(* CODESYS project DCCM_PLC_3_RECOVERED_2023-01-09T10-26-34.project
   Author: jrfsc
   Version: 0.0.0.0
   Title: DCCM_PLC_3

Project tree, tasks and I/O mapping:
  FdtConnections : FDT Connections, Schneider Electric, version 1.0.0.2
  DCCM_PLC_3 : TM251MESC, Schneider Electric, order no. TM251MESC, version 5.1.9.35
      settings: OPCUA enable = False
    application Application
      libraries: SysTimeRtc, * (System); CAA Memory, * (CAA Technical Workgroup); IecRtsServices, 1.0.4.0 (Schneider Electric)
      task MAST (cyclic, interval 20 ms, priority 15, watchdog 100 ms x 1) calls INPUT_MAPPING, AHU_FAN_CONTROL, AHU_DAMPER_CONTROL, AHU_TEMP_CONTROL, RM1_TERMINAL_LOAD, RM2_TERMINAL_LOAD, RM3_TERMINAL_LOAD, RM4_TERMINAL_LOAD, TEST_VAR, SYSTEM_DATE_TIME, OUTPUT_MAPPING, SR_Main
      program AHU_TEMP_CONTROL [FBD]
      program AHU_FAN_CONTROL [FBD]
      program OUTPUT_MAPPING [ST]
      trace Trace (task MAST): GVL.FAN2_SS
      program RM1_TERMINAL_LOAD [FBD]
      global variables PersistentVars
      global variables GVL
      FBs/
        function block DUTY_CHANGE [ST]
        function block LINEAR [ST]
        function block TERMINAL_LOAD [ST]
        function block SB_HEATING_COOLING [ST]
        function block FB_DEPROX_SP [ST]
        function block MAN_AUTO_STS [ST]
        function block FB_HEATING_OR_COOLING [ST]
        function block FB_SETPOINT_MODE [ST]
        function block FB_FLOATING_VALVE [ST]
        function block FB_OMODE [ST]
        function block FB_9StatesMonitoring [ST]
        function block FB_PMODE [ST]
        function block FB_WATCHDOG [ST]
        function block FB_MAX4 [ST]
        function block FB_DUTY_DUTY_STANDBY_PUMP_SPD [ST]
        function block DUTY [ST]
        function block SATSP_CALC [ST]
      program SYSTEM_DATE_TIME [ST]
      program RM3_TERMINAL_LOAD [FBD]
      Library/
        function block FB_SETPOINT_RAMPING [ST]
      program RM2_TERMINAL_LOAD [FBD]
      LIBRARY/
        function block FB_0_10V_TO_2_10V_OUTPUT [ST]
        function block FB_PULSE_GENERATOR [ST]
        function block FB_2_10V_TO_0_10V_INPUT [ST]
      program SR_Main [FBD]
      program AHU_DAMPER_CONTROL [FBD]
      program TEST_VAR [CFC]
      program RM4_TERMINAL_LOAD [FBD]
      program INPUT_MAPPING [ST]
      Enumeration/
        data type ET_9STATE_MONITORING
        data type ET_OMODE
        data type ET_PMODE
    IO_Bus : IO bus - TM3, Schneider Electric, version 5.1.9.35
      Module_3 : TM3AM6/G, Schneider Electric, order no. TM3AM6/G, version 1.0.0.23
          settings: KPI Configuration.KPI Configuration = 32; KPI Configuration.KPI Configuration = 32; KPI Configuration.KPI Configuration = 0; KPI Configuration.KPI Configuration = 0; KPI Configuration.KPI Configuration = 16; KPI Configuration.KPI Configuration = 39; KPI Configuration.KPI Configuration = 16; KPI Configuration.KPI Configuration = 39; KPI Configuration.KPI Configuration = 16; KPI Configuration.KPI Configuration = 16; KPI Configuration.KPI Configuration = 0; KPI Configuration.KPI Configuration = 0; KPI Configuration.KPI Configuration = 16; KPI Configuration.KPI Configuration = 39; KPI Configuration.KPI Configuration = 16; KPI Configuration.KPI Configuration = 39
          input  iOAD1 : INT  // IW0
          input  iOAD2 : INT  // IW1
          output qOAD1 : INT  // QW0
          output qOAD2 : INT  // QW1
          input  ibModule_3_IBStatusIW0 : BYTE  // IBStatusIW0
          input  ibModule_3_IBStatusIW1 : BYTE  // IBStatusIW1
          input  ibModule_3_IBStatusIW2 : BYTE  // IBStatusIW2
          input  ibModule_3_IBStatusIW3 : BYTE  // IBStatusIW3
          input  ibModule_3_IBStatusQW0 : BYTE  // IBStatusQW0
          input  ibModule_3_IBStatusQW1 : BYTE  // IBStatusQW1
          unmapped channels: IW2, IW3
      Module_4 : TM3AM6/G, Schneider Electric, order no. TM3AM6/G, version 1.0.0.23
          settings: KPI Configuration.KPI Configuration = 32; KPI Configuration.KPI Configuration = 32; KPI Configuration.KPI Configuration = 0; KPI Configuration.KPI Configuration = 0; KPI Configuration.KPI Configuration = 16; KPI Configuration.KPI Configuration = 39; KPI Configuration.KPI Configuration = 16; KPI Configuration.KPI Configuration = 39; KPI Configuration.KPI Configuration = 16; KPI Configuration.KPI Configuration = 16; KPI Configuration.KPI Configuration = 0; KPI Configuration.KPI Configuration = 0; KPI Configuration.KPI Configuration = 16; KPI Configuration.KPI Configuration = 39; KPI Configuration.KPI Configuration = 16; KPI Configuration.KPI Configuration = 39
          input  iSAD1_FB : INT  // IW0
          input  iSAD2_FB : INT  // IW1
          output qSAD1 : INT  // QW0
          output qSAD2 : INT  // QW1
          input  ibModule_4_IBStatusIW0 : BYTE  // IBStatusIW0
          input  ibModule_4_IBStatusIW1 : BYTE  // IBStatusIW1
          input  ibModule_4_IBStatusIW2 : BYTE  // IBStatusIW2
          input  ibModule_4_IBStatusIW3 : BYTE  // IBStatusIW3
          input  ibModule_4_IBStatusQW0 : BYTE  // IBStatusQW0
          input  ibModule_4_IBStatusQW1 : BYTE  // IBStatusQW1
          unmapped channels: IW2, IW3
      Module_1 : TM3AM6/G, Schneider Electric, order no. TM3AM6/G, version 1.0.0.23
          settings: KPI Configuration.KPI Configuration = 32; KPI Configuration.KPI Configuration = 32; KPI Configuration.KPI Configuration = 32; KPI Configuration.KPI Configuration = 32; KPI Configuration.KPI Configuration = 0; KPI Configuration.KPI Configuration = 0; KPI Configuration.KPI Configuration = 0; KPI Configuration.KPI Configuration = 0; KPI Configuration.KPI Configuration = 50; KPI Configuration.KPI Configuration = 0; KPI Configuration.KPI Configuration = 244; KPI Configuration.KPI Configuration = 1; KPI Configuration.KPI Configuration = 50; KPI Configuration.KPI Configuration = 0; KPI Configuration.KPI Configuration = 50; KPI Configuration.KPI Configuration = 0; KPI Configuration.KPI Configuration = 200; KPI Configuration.KPI Configuration = 100; KPI Configuration.KPI Configuration = 200; KPI Configuration.KPI Configuration = 200; KPI Configuration.KPI Configuration = 16; KPI Configuration.KPI Configuration = 16; KPI Configuration.KPI Configuration = 0; KPI Configuration.KPI Configuration = 0; KPI Configuration.KPI Configuration = 16; KPI Configuration.KPI Configuration = 39; KPI Configuration.KPI Configuration = 16; KPI Configuration.KPI Configuration = 39
          input  iSA_VELOCITY : INT  // IW0
          input  iFILTER_DP : INT  // IW1
          input  iOA_VELOCITY2 : INT  // IW2
          input  iOA_VELOCITY1 : INT  // IW3
          output qFAN1_SPD : INT  // QW0
          output qFAN2_SPD : INT  // QW1
          input  ibModule_1_IBStatusIW0 : BYTE  // IBStatusIW0
          input  ibModule_1_IBStatusIW1 : BYTE  // IBStatusIW1
          input  ibModule_1_IBStatusIW2 : BYTE  // IBStatusIW2
          input  ibModule_1_IBStatusIW3 : BYTE  // IBStatusIW3
          input  ibModule_1_IBStatusQW0 : BYTE  // IBStatusQW0
          input  ibModule_1_IBStatusQW1 : BYTE  // IBStatusQW1
      Module_6 : TM3TI8T/G, Schneider Electric, order no. TM3TI8T/G, version 1.0.1.21
          settings: KPI Configuration.KPI Configuration = 81; KPI Configuration.KPI Configuration = 81; KPI Configuration.KPI Configuration = 81; KPI Configuration.KPI Configuration = 81; KPI Configuration.KPI Configuration = 81; KPI Configuration.KPI Configuration = 81; KPI Configuration.KPI Configuration = 81; KPI Configuration.KPI Configuration = 81; KPI Configuration.KPI Configuration = 216; KPI Configuration.KPI Configuration = 254; KPI Configuration.KPI Configuration = 216; KPI Configuration.KPI Configuration = 254; KPI Configuration.KPI Configuration = 216; KPI Configuration.KPI Configuration = 254; KPI Configuration.KPI Configuration = 216; KPI Configuration.KPI Configuration = 254; KPI Configuration.KPI Configuration = 216; KPI Configuration.KPI Configuration = 254; KPI Configuration.KPI Configuration = 216; KPI Configuration.KPI Configuration = 254; KPI Configuration.KPI Configuration = 216; KPI Configuration.KPI Configuration = 254; KPI Configuration.KPI Configuration = 216; KPI Configuration.KPI Configuration = 254; KPI Configuration.KPI Configuration = 220; KPI Configuration.KPI Configuration = 5; KPI Configuration.KPI Configuration = 220; KPI Configuration.KPI Configuration = 5; KPI Configuration.KPI Configuration = 220; KPI Configuration.KPI Configuration = 5; KPI Configuration.KPI Configuration = 220; KPI Configuration.KPI Configuration = 5; KPI Configuration.KPI Configuration = 220; KPI Configuration.KPI Configuration = 5; KPI Configuration.KPI Configuration = 220; KPI Configuration.KPI Configuration = 5; KPI Configuration.KPI Configuration = 220; KPI Configuration.KPI Configuration = 5; KPI Configuration.KPI Configuration = 220; KPI Configuration.KPI Configuration = 5;
            KPI Configuration.KPI Configuration = 16; KPI Configuration.KPI Configuration = 39; KPI Configuration.KPI Configuration = 137; KPI Configuration.KPI Configuration = 15; KPI Configuration.KPI Configuration = 16; KPI Configuration.KPI Configuration = 39; KPI Configuration.KPI Configuration = 137; KPI Configuration.KPI Configuration = 15; KPI Configuration.KPI Configuration = 16; KPI Configuration.KPI Configuration = 39; KPI Configuration.KPI Configuration = 137; KPI Configuration.KPI Configuration = 15; KPI Configuration.KPI Configuration = 16; KPI Configuration.KPI Configuration = 39; KPI Configuration.KPI Configuration = 137; KPI Configuration.KPI Configuration = 15; KPI Configuration.KPI Configuration = 16; KPI Configuration.KPI Configuration = 39; KPI Configuration.KPI Configuration = 137; KPI Configuration.KPI Configuration = 15; KPI Configuration.KPI Configuration = 16; KPI Configuration.KPI Configuration = 39; KPI Configuration.KPI Configuration = 137; KPI Configuration.KPI Configuration = 15; KPI Configuration.KPI Configuration = 16; KPI Configuration.KPI Configuration = 39; KPI Configuration.KPI Configuration = 137; KPI Configuration.KPI Configuration = 15; KPI Configuration.KPI Configuration = 16; KPI Configuration.KPI Configuration = 39; KPI Configuration.KPI Configuration = 137; KPI Configuration.KPI Configuration = 15
          input  iSAT : INT  // IW0
          input  iRAT : INT  // IW1
          input  iOCT : INT  // IW2
          input  iOAT : INT  // IW3
          input  iRMT1 : INT  // IW4
          input  iRMT2 : INT  // IW5
          input  iRMT3 : INT  // IW6
          input  iRMT4 : INT  // IW7
          input  ibModule_6_IBStatusIW0 : BYTE  // IBStatusIW0
          input  ibModule_6_IBStatusIW1 : BYTE  // IBStatusIW1
          input  ibModule_6_IBStatusIW2 : BYTE  // IBStatusIW2
          input  ibModule_6_IBStatusIW3 : BYTE  // IBStatusIW3
          input  ibModule_6_IBStatusIW4 : BYTE  // IBStatusIW4
          input  ibModule_6_IBStatusIW5 : BYTE  // IBStatusIW5
          input  ibModule_6_IBStatusIW6 : BYTE  // IBStatusIW6
          input  ibModule_6_IBStatusIW7 : BYTE  // IBStatusIW7
      Module_2 : TM3AM6/G, Schneider Electric, order no. TM3AM6/G, version 1.0.0.23
          settings: KPI Configuration.KPI Configuration = 32; KPI Configuration.KPI Configuration = 32; KPI Configuration.KPI Configuration = 32; KPI Configuration.KPI Configuration = 0; KPI Configuration.KPI Configuration = 0; KPI Configuration.KPI Configuration = 0; KPI Configuration.KPI Configuration = 16; KPI Configuration.KPI Configuration = 39; KPI Configuration.KPI Configuration = 16; KPI Configuration.KPI Configuration = 39; KPI Configuration.KPI Configuration = 244; KPI Configuration.KPI Configuration = 1; KPI Configuration.KPI Configuration = 200; KPI Configuration.KPI Configuration = 16; KPI Configuration.KPI Configuration = 16; KPI Configuration.KPI Configuration = 0; KPI Configuration.KPI Configuration = 0; KPI Configuration.KPI Configuration = 16; KPI Configuration.KPI Configuration = 39; KPI Configuration.KPI Configuration = 16; KPI Configuration.KPI Configuration = 39
          input  iFAN1_SPDFB : INT  // IW0
          input  iFAN2_SPDFB : INT  // IW1
          input  iFILTER2_DP : INT  // IW2
          output qAHU_HV : INT  // QW0
          output qAHU_CV : INT  // QW1
          input  ibModule_2_IBStatusIW0 : BYTE  // IBStatusIW0
          input  ibModule_2_IBStatusIW1 : BYTE  // IBStatusIW1
          input  ibModule_2_IBStatusIW2 : BYTE  // IBStatusIW2
          input  ibModule_2_IBStatusIW3 : BYTE  // IBStatusIW3
          input  ibModule_2_IBStatusQW0 : BYTE  // IBStatusQW0
          input  ibModule_2_IBStatusQW1 : BYTE  // IBStatusQW1
          unmapped channels: IW3
      Module_5 : TM3DM24R/G, Schneider Electric, order no. TM3DM24R/G, version 1.0.2.0
          input  iFAN1_RUN : BOOL  // IW0.I0
          input  iFAN1_FAULT : BOOL  // IW0.I1
          input  iFAN1_READY : BOOL  // IW0.I2
          input  iFAN2_RUN : BOOL  // IW0.I3
          input  iFAN2_FAULT : BOOL  // IW0.I4
          input  iFAN2_READY : BOOL  // IW0.I5
          input  iRAD1_2_STS : BOOL  // IW0.I6
          input  iFIRE_DAMPER_STS : BOOL  // IW0.I7
          input  iDUCT_SMOKE_DETECTOR : BOOL  // IW0.I8
          input  iFAN1_MANUAL_SW : BOOL  // IW0.I12
          input  iFAN1_AUTO_SW : BOOL  // IW0.I13
          input  iFAN2_MANUAL_SW : BOOL  // IW0.I14
          input  iFAN2_AUTO_SW : BOOL  // IW0.I15
          output qFAN1_SS : BOOL  // QB0.Q0
          output qFAN2_SS : BOOL  // QB0.Q1
          output qFAN1_RAD1_2 : BOOL  // QB0.Q2
          output qISO_NORMAL_MODE : BOOL  // QB0.Q3
          unmapped channels: IW0, QB0
    Serial_Line_1 : Serial line, Schneider Electric, version 5.1.9.35
      Machine_Expert_Network_Manager : Machine Expert-Network Manager, Schneider Electric, version 4.0.0.4
    CAN_1 : CANopen bus, Schneider Electric, version 5.1.9.35
    COM_Bus : COM bus, Schneider Electric, version 5.1.9.35
    Ethernet_1 : Ethernet Network, Schneider Electric, version 5.1.9.35
        settings: WebServer = TRUE; FTP Server = FALSE; SoMachine Protocol = TRUE; Modbus Server = TRUE; NetManage Protocol = TRUE; SNMP protocol = FALSE; WebVisu protocol = FALSE; Secured Web Server = TRUE
*)

// DCCM_PLC_3/Application/Enumeration/ET_9STATE_MONITORING
{attribute 'qualified_only' := ''}
{attribute 'strict' := ''}
TYPE ET_9STATE_MONITORING :
(
	STOPPED := 0,
	RUNNING := 1,
	STARTING := 2,
	STOPPING := 3,
	START_FAIL := 4,
	STOP_FAIL := 5,
	UNEXPECTED_START := 6,
	UNEXPECTED_STOP := 7,
	FIRE_STOP := 8,
	UNKNOWN := 9
);
END_TYPE

// DCCM_PLC_3/Application/Enumeration/ET_OMODE
{attribute 'qualified_only' := ''}
{attribute 'strict' := ''}
TYPE ET_OMODE :
(
	UNOCC := 0,
	OPTSTART := 1,
	SCH := 2,
	AHRS := 3,
	MOTDETECT := 4,
	SETBACK := 7
);
END_TYPE

// DCCM_PLC_3/Application/Enumeration/ET_PMODE
{attribute 'qualified_only' := ''}
{attribute 'strict' := ''}
TYPE ET_PMODE :
(
	OFF_NORMAL := 0,
	OFF_PCMS := 1,
	OFF_Fire := 2,
	OFF_DMPRLOCK := 3,
	OFF_RESET := 4,
	Startup := 5,
	Purge := 6,
	RUN_NORMAL := 7
);
END_TYPE

// DCCM_PLC_3/Application/PersistentVars
{attribute 'qualified_only'}
VAR_GLOBAL PERSISTENT RETAIN
	// Generated instance path of persistent variable
	GVL.RM1_RMTSP: REAL := 22.0;
	// Generated instance path of persistent variable
	GVL.RM2_RMTSP: REAL := 22.0;
	// Generated instance path of persistent variable
	GVL.RM3_RMTSP: REAL := 22.0;
	// Generated instance path of persistent variable
	GVL.FAN1_SPD_MAN: REAL;
	// Generated instance path of persistent variable
	GVL.SA_VELOCITY_SP: REAL := 35.0;
	// Generated instance path of persistent variable
	GVL.FILTER_DPSP: REAL := 100.0;
	// Generated instance path of persistent variable
	GVL.SATSP_MAX: REAL := 30.0;
	// Generated instance path of persistent variable
	GVL.SATSP_MIN: REAL := 12.0;
	// Generated instance path of persistent variable
	GVL.SATSP_MID: REAL := 20.0;
	// Generated instance path of persistent variable
	GVL.AHU_POAD_SP: REAL := 0.0;
	// Generated instance path of persistent variable
	GVL.AHU_OAD_SP: REAL := 100.0;
	// Generated instance path of persistent variable
	GVL.FILTER2_DP_ALMSP: REAL := 350.0;
	// Generated instance path of persistent variable
	GVL.FAN_DEPROX1_SP: REAL := 18.0;
	// Generated instance path of persistent variable
	GVL.FAN_DEPROX2_SP: REAL := 1.0;
	// Generated instance path of persistent variable
	GVL.FAN_DEPROX4_SPDSP: REAL := 0.0;
	// Generated instance path of persistent variable
	GVL.FAN_DEPROX4_SP: REAL := 0.0;
END_VAR

// DCCM_PLC_3/Application/GVL
{attribute 'qualified_only'}
VAR_GLOBAL
	AHU_RAD_MAN AT %MD550: REAL;
	AHU_RAD_MD AT %MX5.6: bool;
	FAN1_SPD AT %MD500: REAL;
	FAN2_SPD AT %MD501: REAL;
	SA_VELOCITY AT %MD502: REAL;
	FILTER_DP AT %MD503: REAL;
	OA_VELOCITY1 AT %MD504: REAL;
	OA_VELOCITY2 AT %MD505: REAL;
	AHU_HV AT %MD506: REAL;
	AHU_CV AT %MD507: REAL;
	FAN1_SPDFB AT %MD508: REAL;
	FAN2_SPDFB AT %MD509: REAL;
	OAD AT %MD510: REAL;
	SAD1 AT %MD512: REAL;
	SAD2 AT %MD513: REAL;
	FAN1_RUN AT %MX0.0: BOOL;
	FAN1_FAULT AT %MX0.1: BOOL;
	FAN1_READY AT %MX0.2: BOOL;
	FAN2_RUN AT %MX0.3: BOOL;
	FAN2_FAULT AT %MX0.4: BOOL;
	FAN2_READY AT %MX0.5: BOOL;
	RAD1_2_STS AT %MX0.6: BOOL;
	FIRE_DAMPER_STS AT %MX0.7: BOOL;
	DUCT_SMOKE_DETECTOR AT %MX1.0: BOOL;
	FAN1_MANUAL_SW AT %MX1.1: BOOL;
	FAN1_AUTO_SW AT %MX1.2: BOOL;
	FAN2_MANUAL_SW AT %MX1.3: BOOL;
	FAN2_AUTO_SW AT %MX1.4: BOOL;
	FAN1_SS AT %MX1.5: BOOL;
	FAN2_SS AT %MX1.6: BOOL;
	FAN1_RAD1_2 AT %MX1.7: BOOL;
	// NEED TO FIGURE OUT WHAT THIS DOES
	ISO_NORMAL_MODE AT %MX2.0: BOOL;
	SAT AT %MD514: REAL;
	RAT AT %MD515: REAL;
	OCT AT %MD516: REAL;
	OAT AT %MD517: REAL;
	RMT1 AT %MD518: REAL;
	RMT2 AT %MD519: REAL;
	RMT3 AT %MD520: REAL;
	RMT4 AT %MD521: REAL;
END_VAR
VAR_GLOBAL RETAIN PERSISTENT
	RM1_RMTSP AT %MD522: REAL := 22;
	RM2_RMTSP AT %MD523: REAL := 22;
	RM3_RMTSP AT %MD524: REAL := 22;
END_VAR
VAR_GLOBAL RETAIN
	RM4_RMTSP AT %MD525: REAL := 22;
END_VAR
VAR_GLOBAL PERSISTENT
	FAN1_SPD_MAN AT %MD526: REAL;
END_VAR
VAR_GLOBAL
	FAN1_SPD_MD AT %MX2.1: BOOL := TRUE;
	FAN2_SPD_MAN AT %MD527: REAL;
	FAN2_SPD_MD AT %MX2.2: BOOL := TRUE;
END_VAR
VAR_GLOBAL RETAIN PERSISTENT
	SA_VELOCITY_SP AT %MD528: REAL := 35;
	FILTER_DPSP AT %MD529: REAL := 100;
END_VAR
VAR_GLOBAL
	FILTER_DP_ALM AT %MX2.3: BOOL;
	AHU_HV_MAN AT %MD530: REAL;
	AHU_HV_MD AT %MX2.4: BOOL := TRUE;
	AHU_CV_MAN AT %MD531: REAL;
	AHU_CV_MD AT %MX2.5: BOOL := TRUE;
	OAD_MAN AT %MD532: REAL;
	OAD_MD AT %MX2.6: BOOL := TRUE;
	SAD1_MAN AT %MD534: REAL;
	SAD1_MD AT %MX3.0: BOOL := TRUE;
	SAD2_MAN AT %MD535: REAL;
	SAD2_MD AT %MX3.1: BOOL := TRUE;
	FAN1_SS_MAN AT %MX3.2: BOOL;
	FAN1_SS_MD AT %MX3.3: BOOL := TRUE;
	FAN2_SS_MAN AT %MX3.4: BOOL;
	FAN2_SS_MD AT %MX3.5: BOOL := TRUE;
	RM1_TL AT %MD536: REAL;
	RM2_TL AT %MD537: REAL;
	RM3_TL AT %MD538: REAL;
	RM4_TL AT %MD539: REAL;
	TL AT %MD540: REAL;
	SATSP AT %MD541: REAL;
	SATSP_MAN AT %MD542: REAL;
	SATSP_MD AT %MX3.6: BOOL := TRUE;
END_VAR
VAR_GLOBAL RETAIN PERSISTENT
	SATSP_MAX AT %MD543: REAL := 30;
	SATSP_MIN AT %MD544: REAL := 12;
END_VAR
VAR_GLOBAL
	FAN_DUTY AT %MX3.7: BOOL;
	FAN_DUTY_MAN AT %MX4.0: BOOL;
	FAN_DUTY_MD AT %MX4.1: BOOL := TRUE;
	SYS_DAY: UINT;
	SYS_HOUR: UINT;
	SYS_MINUTE: UINT;
	FAN1_STS AT %MW9000: UINT;
	FAN2_STS AT %MW9001: UINT;
	FAN1_RAD1_2_MAN AT %MX6.4: BOOL;
	FAN1_RAD1_2_MD AT %MX4.2: BOOL := TRUE;
	MAX_TL AT %MD546: REAL;
	FAN2_DISCHARGE_DAMPER AT %MX5.3: BOOL;
END_VAR
VAR_GLOBAL RETAIN PERSISTENT
	SATSP_MID AT %MD547: REAL := 20;
END_VAR
VAR_GLOBAL
	PANDEMIC_MODE AT %MX4.3: BOOL;
	FAN1_DISCHARGE_DAMPER AT %MX5.0: BOOL;
	FAN1_DISCHARGE_DAMPER_MD AT %MX5.1: BOOL := TRUE;
	FAN2_DISCHARGE_DAMPER_MD AT %MX5.4: BOOL := TRUE;
	FAN2_DISCHARGE_DAMPER_MAN AT %MX5.5: BOOL;
	FAN1_DISCHARGE_DAMPER_MAN AT %MX5.2: BOOL;
	EAD AT %MD548: REAL;
	AHU_RAD AT %MD549: REAL;
	FAN1_DISCHARGE_DAMPER_STS AT %MX5.7: BOOL;
	FAN2_DISCHARGE_DAMPER_STS AT %MX6.0: BOOL;
	POAD_MAN AT %MD559: REAL;
END_VAR
VAR_GLOBAL RETAIN PERSISTENT
	AHU_POAD_SP AT %MD554: REAL := 0;
END_VAR
VAR_GLOBAL
	POAD_MD AT %MX6.2: BOOL := TRUE;
	POAD AT %MD555: REAL;
	OAD_VELOCITY AT %MD556: REAL;
	OAP_VELOCITY AT %MD557: REAL;
	OAD_STS AT %MD560: REAL;
	OAP_STS AT %MD561: REAL;
END_VAR
VAR_GLOBAL RETAIN PERSISTENT
	AHU_OAD_SP AT %MD558: REAL := 100;
END_VAR
VAR_GLOBAL
	FAN1_DAMPER_STS AT %MD562: REAL;
	FAN2_DAMPER_STS AT %MD563: REAL;
	OAD1_FB AT %MD550: REAL;
	OAD2_FB AT %MD551: REAL;
	SAD1_FB AT %MD552: REAL;
	SAD2_FB AT %MD553: REAL;
	PAN_MODE_OK AT %MX6.1: BOOL;
	OAD_LS AT %MD564: REAL;
	POAD_LS AT %MD565: REAL;
	SAD_LS AT %MD566: REAL;
	FAN1_SW_STS AT %MW9002: INT;
	FAN2_SW_STS AT %MW9003: INT;
	FILTER2_DP AT %MD567: REAL;
END_VAR
VAR_GLOBAL RETAIN PERSISTENT
	FILTER2_DP_ALMSP AT %MD568: REAL := 350;
END_VAR
VAR_GLOBAL
	FILTER2_DP_ALM AT %MX6.3: BOOL;
END_VAR
VAR_GLOBAL RETAIN PERSISTENT
	FAN_DEPROX1_SP AT %MD569: REAL := 18;
	FAN_DEPROX2_SP AT %MD570: REAL := 1;
	FAN_DEPROX4_SPDSP AT %MD571: REAL := 0;
END_VAR
VAR_GLOBAL
	ROOM1_DEPROX: INT;
	ROOM2_DEPROX: INT;
	ROOM3_DEPROX: INT;
	ROOM4_DEPROX: INT;
END_VAR
VAR_GLOBAL RETAIN PERSISTENT
	FAN_DEPROX4_SP AT %MD571: REAL := 0;
END_VAR
VAR_GLOBAL
	SAD1_ALM AT %MX6.4: BOOL;
	SAD2_ALM AT %MX6.5: BOOL;
	OAD_ALM AT %MX6.6: BOOL;
	POAD_ALM AT %MX6.7: BOOL;
	RAD_ALM AT %MX7.0: BOOL;
	PAND_ALM AT %MX7.1: BOOL;
	SEND_PAND_ALM AT %MW9004: INT;
	OAD_L2_SP AT %MD572: REAL;
	POAD_L2_SP AT %MD573: REAL;
	SA_L2_SP AT %MD574: REAL;
	FAN1_DIG_FLT AT %MX7.2: BOOL;
	FAN2_DIG_FLT AT %MX7.3: BOOL;
	FAN2_FLT_RESET AT %MX7.4: BOOL;
	FAN1_FLT_RESET AT %MX7.5: BOOL;
END_VAR

// DCCM_PLC_3/Application/INPUT_MAPPING
PROGRAM INPUT_MAPPING
VAR
	BELIMO_IP: FB_2_10V_TO_0_10V_INPUT;
END_VAR

//MAPPING HARDWARE INPUTS TO MEMORY WORDS

GVL.SA_VELOCITY := TO_REAL(iSA_VELOCITY);					//MODULE 1 TM3AM6 INPUT 0
GVL.FILTER_DP := TO_REAL(iFILTER_DP);						//MODULE 1 TM3AM6 INPUT 1
//GVL.OA_VELOCITY1 := TO_REAL(iOA_VELOCITY1);	LOOK AT BOTTOM OF MAPPING				//MODULE 1 TM3AM6 INPUT 2
//GVL.OA_VELOCI0TY2 := TO_REAL(iOA_VELOCITY2);					//MODULE 1 TM3AM6 INPUT 3

GVL.FAN1_SPDFB := TO_REAL(iFAN1_SPDFB) / 100;						//MODULE 2 TM3AM6 INPUT 0
GVL.FAN2_SPDFB := TO_REAL(iFAN2_SPDFB) / 100;						//MODULE 2 TM3AM6 INPUT 1

//GVL.OAD1_FB := TO_REAL(iOAD1);		 LOOK AT BOTTOM OF MAPPING		//MODULE 3 TM3AM6 INPUT 0
//GVL.OAD2_FB := TO_REAL(iOAD2);								//MODULE 3 TM3AM6 INPUT 1

GVL.SAD1_FB := TO_REAL(iSAD1_FB);							//MODULE 4 TM3AM6 INPUT 0
GVL.SAD2_FB := TO_REAL(iSAD2_FB);							//MODULE 4 TM3AM6 INPUT 1

GVL.FAN1_RUN := iFAN1_RUN;									//MODULE 5 TM3DM24R INPUT 0
GVL.FAN1_FAULT := iFAN1_FAULT;								//MODULE 5 TM3DM24R INPUT 1
GVL.FAN1_READY := iFAN1_READY;								//MODULE 5 TM3DM24R INPUT 2
GVL.FAN2_RUN := iFAN2_RUN;									//MODULE 5 TM3DM24R INPUT 3
GVL.FAN2_FAULT := iFAN2_FAULT;								//MODULE 5 TM3DM24R INPUT 4
GVL.FAN2_READY := iFAN2_READY;								//MODULE 5 TM3DM24R INPUT 5
GVL.RAD1_2_STS := NOT(iRAD1_2_STS);								//MODULE 5 TM3DM24R INPUT 6
GVL.FIRE_DAMPER_STS := iFIRE_DAMPER_STS;					//MODULE 5 TM3DM24R INPUT 7
GVL.DUCT_SMOKE_DETECTOR := iDUCT_SMOKE_DETECTOR;			//MODULE 5 TM3DM24R INPUT 8

GVL.FAN1_MANUAL_SW := iFAN1_MANUAL_SW;						//MODULE 5 TM3DM24R INPUT 12
GVL.FAN1_AUTO_SW := iFAN1_AUTO_SW;							//MODULE 5 TM3DM24R INPUT 13
GVL.FAN2_MANUAL_SW := iFAN2_MANUAL_SW;						//MODULE 5 TM3DM24R INPUT 14
GVL.FAN2_AUTO_SW := iFAN2_AUTO_SW;							//MODULE 5 TM3DM24R INPUT 15

GVL.SAT := TO_REAL(iSAT) / 10.0;											//MODULE 6 TM3TI8T INPUT 0
GVL.RAT := TO_REAL(iRAT) / 10.0;											//MODULE 6 TM3TI8T INPUT 1
GVL.OCT := TO_REAL(iOCT) / 10.0;											//MODULE 6 TM3TI8T INPUT 2
GVL.OAT := TO_REAL(iOAT) / 10.0;											//MODULE 6 TM3TI8T INPUT 3
GVL.RMT1 := TO_REAL(iRMT1) / 10.0;											//MODULE 6 TM3TI8T INPUT 4
GVL.RMT2 := TO_REAL(iRMT2) / 10.0;											//MODULE 6 TM3TI8T INPUT 5
GVL.RMT3 := TO_REAL(iRMT3) / 10.0;											//MODULE 6 TM3TI8T INPUT 6
GVL.RMT4 := TO_REAL(iRMT4) / 10.0;											//MODULE 6 TM3TI8T INPUT 7

//To be assigned
GVL.OAD_VELOCITY := TO_REAL(iOA_VELOCITY1);	 //Outside Air Velocity from OA Damper
GVL.OAP_VELOCITY := TO_REAL(iOA_VELOCITY2);	 //Outside Air Velocity from OA Pandemic Mode Damper
BELIMO_IP(IN_PRCT := (TO_REAL(iOAD1) / 100));
GVL.OAD_STS := 100 - BELIMO_IP.OUT_PRCT;				 //OA Damper FEEDBACK
BELIMO_IP(IN_PRCT := (TO_REAL(iOAD2) / 100));
GVL.OAP_STS := 100 - BELIMO_IP.OUT_PRCT;			     //OA Pandemic Mode Damper FEEDBACK

BELIMO_IP(IN_PRCT := TO_REAL(iSAD1_FB) / 100);
GVL.FAN1_DAMPER_STS := 100 - BELIMO_IP.OUT_PRCT;	//FAN1 Damper
BELIMO_IP(IN_PRCT := TO_REAL(iSAD2_FB) / 100);
GVL.FAN2_DAMPER_STS := 100 - BELIMO_IP.OUT_PRCT;	//FAN2 Damper

GVL.FILTER2_DP := TO_REAL(iFILTER2_DP);				//SECOND FILTER DP

GVL.OAD_LS := GVL.OAD_VELOCITY * 19.5;					//OAD VP IN L/S
GVL.POAD_LS := GVL.OAP_VELOCITY * 63;				//OAP VP IN L/S
GVL.SAD_LS := GVL.SA_VELOCITY * 25.21;						//SAD VP L/S

GVL.SEND_PAND_ALM := TO_INT(GVL.PANDEMIC_MODE);


GVL.SA_L2_SP := GVL.SA_VELOCITY_SP * 25.21;

END_PROGRAM

// DCCM_PLC_3/Application/LIBRARY/FB_2_10V_TO_0_10V_INPUT
FUNCTION_BLOCK FB_2_10V_TO_0_10V_INPUT
VAR_INPUT
	/// 0-10V = 0-100%
	IN_PRCT: REAL;
END_VAR
VAR_OUTPUT
	/// 2-10V = 0-100%
	OUT_PRCT: REAL;
END_VAR
VAR
	result: REAL;
	LIN: LINEAR;
END_VAR

LIN (X1:=2, Y1:=0, X2:=10, Y2:=10, INPUT:= IN_PRCT/10);
OUT_PRCT := MAX(0, MIN(LIN.OUTPUT * 10, 100));

END_FUNCTION_BLOCK

// DCCM_PLC_3/Application/FBs/LINEAR
FUNCTION_BLOCK LINEAR
VAR_INPUT
	INPUT: REAL;
	X1: REAL;
	Y1: REAL;
	X2: REAL;
	Y2: REAL;
END_VAR
VAR
	M: REAL;
END_VAR
VAR_OUTPUT
	OUTPUT: REAL;
END_VAR

// Y1-Y2 = M(X1-X2)
//M = (Y2-Y1)/(X2-X1)

M := (Y2 - Y1) / (X2 - X1);
OUTPUT := (M * (INPUT - X1)) + Y1;

END_FUNCTION_BLOCK

// DCCM_PLC_3/Application/AHU_FAN_CONTROL
PROGRAM AHU_FAN_CONTROL
VAR
	DUTY_CHANGE_0: DUTY_CHANGE;
	FB_9StatesMonitoring_0: FB_9StatesMonitoring;
	FB_9StatesMonitoring_1: FB_9StatesMonitoring;
	SPD_PID: PID;
	SPD: REAL;
	SPD_P: REAL := 1.5;
	SPD_I: REAL := 250;
	TON_0: TON;
	LINEAR_0: LINEAR;
	A: BOOL;
	LINEAR_1: LINEAR;
	B: BOOL;
	MAN_AUTO_STS_0: MAN_AUTO_STS;
	MAN_AUTO_STS_1: MAN_AUTO_STS;
	FB_DEPROX_SP_0: FB_DEPROX_SP;
	TEMP_SP: REAL;
	RM_TTL: REAL;
	SAD_FB_SP: REAL := 90;
	OUTSIDE_DAMPER_OK: BOOL;
	TON_1: TON;
	TON_2: TON;
	RS_0: RS;
	RS_1: RS;
	FAN1_FLT_RESET: BOOL;
	FAN2_FLT_RESET: BOOL;
END_VAR

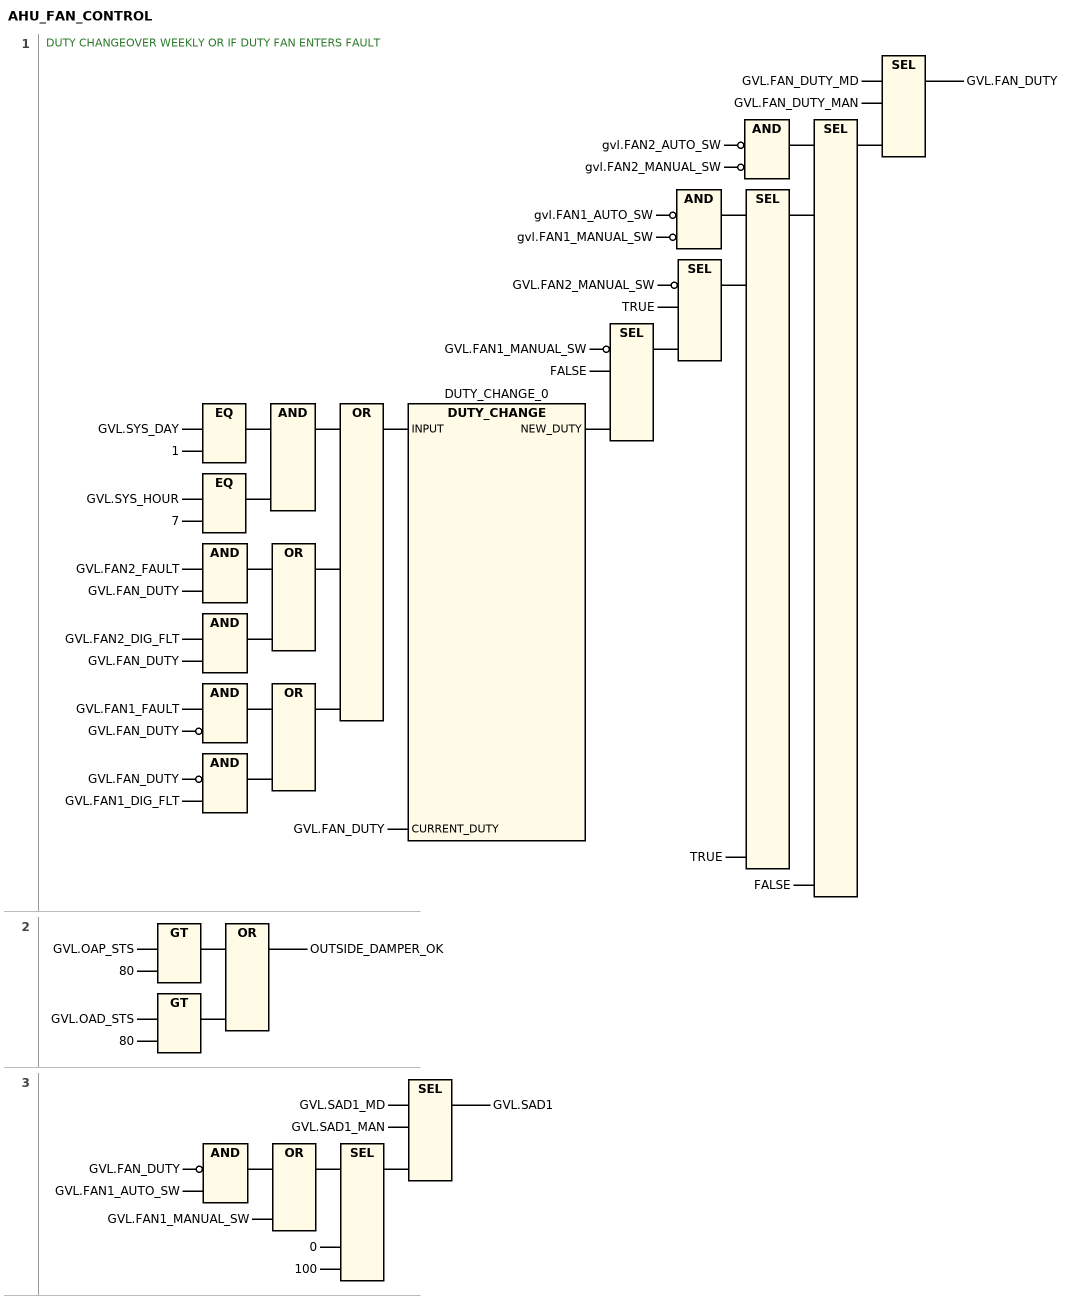
// NETWORK 1
// DUTY CHANGEOVER WEEKLY OR IF DUTY FAN ENTERS FAULT
DUTY_CHANGE_0(INPUT := GVL.SYS_DAY = 1 AND GVL.SYS_HOUR = 7 OR (GVL.FAN2_FAULT AND GVL.FAN_DUTY OR GVL.FAN2_DIG_FLT AND GVL.FAN_DUTY) OR (GVL.FAN1_FAULT AND NOT GVL.FAN_DUTY OR NOT GVL.FAN_DUTY AND GVL.FAN1_DIG_FLT), CURRENT_DUTY := GVL.FAN_DUTY); // DUTY_CHANGE
GVL.FAN_DUTY := SEL(GVL.FAN_DUTY_MD, GVL.FAN_DUTY_MAN, SEL(NOT gvl.FAN2_AUTO_SW AND NOT gvl.FAN2_MANUAL_SW, SEL(NOT gvl.FAN1_AUTO_SW AND NOT gvl.FAN1_MANUAL_SW, SEL(NOT GVL.FAN2_MANUAL_SW, TRUE, SEL(NOT GVL.FAN1_MANUAL_SW, FALSE, DUTY_CHANGE_0.NEW_DUTY)), TRUE), FALSE));

// NETWORK 2
OUTSIDE_DAMPER_OK := GVL.OAP_STS > 80 OR GVL.OAD_STS > 80;

// NETWORK 3
GVL.SAD1 := SEL(GVL.SAD1_MD, GVL.SAD1_MAN, SEL(NOT GVL.FAN_DUTY AND GVL.FAN1_AUTO_SW OR GVL.FAN1_MANUAL_SW, 0, 100));

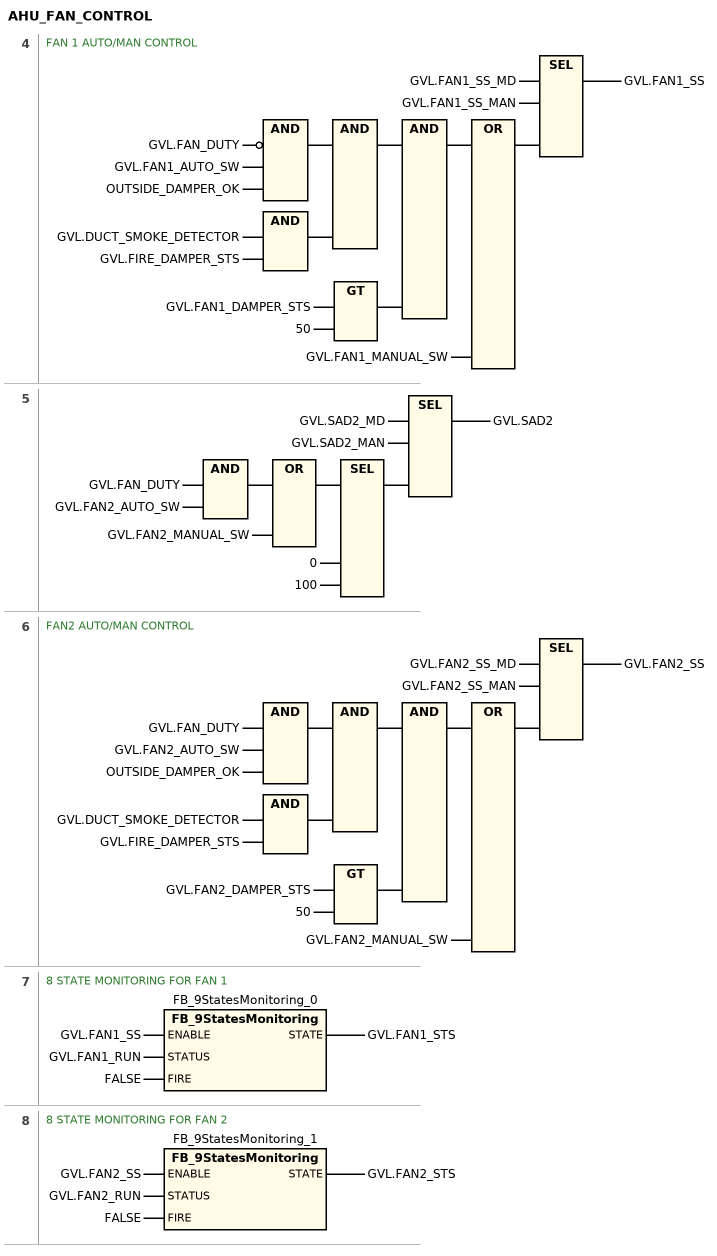
// NETWORK 4
// FAN 1 AUTO/MAN CONTROL
GVL.FAN1_SS := SEL(GVL.FAN1_SS_MD, GVL.FAN1_SS_MAN, ((NOT GVL.FAN_DUTY AND GVL.FAN1_AUTO_SW AND OUTSIDE_DAMPER_OK) AND (GVL.DUCT_SMOKE_DETECTOR AND GVL.FIRE_DAMPER_STS)) AND GVL.FAN1_DAMPER_STS > 50 OR GVL.FAN1_MANUAL_SW);

// NETWORK 5
GVL.SAD2 := SEL(GVL.SAD2_MD, GVL.SAD2_MAN, SEL(GVL.FAN_DUTY AND GVL.FAN2_AUTO_SW OR GVL.FAN2_MANUAL_SW, 0, 100));

// NETWORK 6
// FAN2 AUTO/MAN CONTROL
GVL.FAN2_SS := SEL(GVL.FAN2_SS_MD, GVL.FAN2_SS_MAN, ((GVL.FAN_DUTY AND GVL.FAN2_AUTO_SW AND OUTSIDE_DAMPER_OK) AND (GVL.DUCT_SMOKE_DETECTOR AND GVL.FIRE_DAMPER_STS)) AND GVL.FAN2_DAMPER_STS > 50 OR GVL.FAN2_MANUAL_SW);

// NETWORK 7
// 8 STATE MONITORING FOR FAN 1
FB_9StatesMonitoring_0(ENABLE := GVL.FAN1_SS, STATUS := GVL.FAN1_RUN, FIRE := FALSE); // FB_9StatesMonitoring
GVL.FAN1_STS := FB_9StatesMonitoring_0.STATE;

// NETWORK 8
// 8 STATE MONITORING FOR FAN 2
FB_9StatesMonitoring_1(ENABLE := GVL.FAN2_SS, STATUS := GVL.FAN2_RUN, FIRE := FALSE); // FB_9StatesMonitoring
GVL.FAN2_STS := FB_9StatesMonitoring_1.STATE;

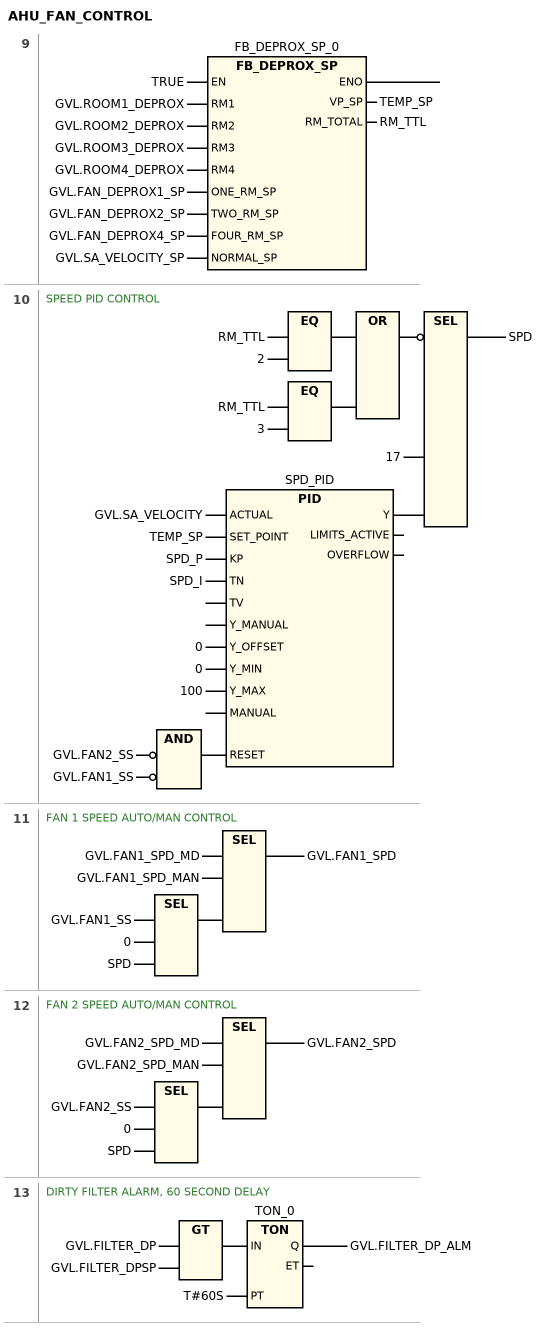
// NETWORK 9
FB_DEPROX_SP_0(
    RM1 := GVL.ROOM1_DEPROX,
    RM2 := GVL.ROOM2_DEPROX,
    RM3 := GVL.ROOM3_DEPROX,
    RM4 := GVL.ROOM4_DEPROX,
    ONE_RM_SP := GVL.FAN_DEPROX1_SP,
    TWO_RM_SP := GVL.FAN_DEPROX2_SP,
    FOUR_RM_SP := GVL.FAN_DEPROX4_SP,
    NORMAL_SP := GVL.SA_VELOCITY_SP,
    VP_SP => TEMP_SP,
    RM_TOTAL => RM_TTL); // FB_DEPROX_SP

// NETWORK 10
// SPEED PID CONTROL
SPD_PID(
    ACTUAL := GVL.SA_VELOCITY,
    SET_POINT := TEMP_SP,
    KP := SPD_P,
    TN := SPD_I,
    Y_OFFSET := 0,
    Y_MIN := 0,
    Y_MAX := 100,
    RESET := NOT GVL.FAN2_SS AND NOT GVL.FAN1_SS); // PID
SPD := SEL(NOT (RM_TTL = 2 OR RM_TTL = 3), 17, SPD_PID.Y);

// NETWORK 11
// FAN 1 SPEED AUTO/MAN CONTROL
GVL.FAN1_SPD := SEL(GVL.FAN1_SPD_MD, GVL.FAN1_SPD_MAN, SEL(GVL.FAN1_SS, 0, SPD));

// NETWORK 12
// FAN 2 SPEED AUTO/MAN CONTROL
GVL.FAN2_SPD := SEL(GVL.FAN2_SPD_MD, GVL.FAN2_SPD_MAN, SEL(GVL.FAN2_SS, 0, SPD));

// NETWORK 13
// DIRTY FILTER ALARM, 60 SECOND DELAY
TON_0(IN := GVL.FILTER_DP > GVL.FILTER_DPSP, PT := T#60S); // TON
GVL.FILTER_DP_ALM := TON_0.Q;

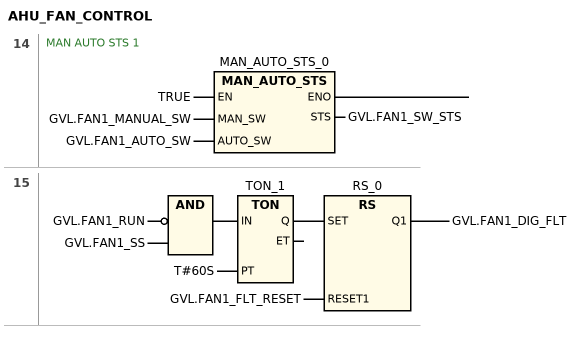
// NETWORK 14
// MAN AUTO STS 1
MAN_AUTO_STS_0(MAN_SW := GVL.FAN1_MANUAL_SW, AUTO_SW := GVL.FAN1_AUTO_SW, STS => GVL.FAN1_SW_STS); // MAN_AUTO_STS

// NETWORK 15
TON_1(IN := NOT GVL.FAN1_RUN AND GVL.FAN1_SS, PT := T#60S); // TON
RS_0(SET := TON_1.Q, RESET1 := GVL.FAN1_FLT_RESET); // RS
GVL.FAN1_DIG_FLT := RS_0.Q1;

END_PROGRAM

// DCCM_PLC_3/Application/FBs/DUTY_CHANGE
FUNCTION_BLOCK DUTY_CHANGE
VAR_INPUT
	INPUT: BOOL;
END_VAR
VAR_OUTPUT
	NEW_DUTY: BOOL;
END_VAR
VAR_INPUT
	CURRENT_DUTY: BOOL;
END_VAR

IF INPUT THEN
	IF CURRENT_DUTY = 1 THEN
		NEW_DUTY := 0;
	ELSIF CURRENT_DUTY = 0 THEN
		NEW_DUTY := 1;
	END_IF
END_IF

END_FUNCTION_BLOCK

// DCCM_PLC_3/Application/FBs/FB_9StatesMonitoring
FUNCTION_BLOCK FB_9StatesMonitoring
VAR
	ENABLE_OFF: BOOL := FALSE;
	ENABLE_ON: BOOL := FALSE;
	STATUS_ON: BOOL := FALSE;
	STATUS_OFF: BOOL := FALSE;
	FIRE_ON: BOOL := FALSE;
	FIRE_OFF: BOOL := FALSE;
	BEEN_RUNNING_OK: BOOL := FALSE;
	NOT_BEEN_RUNNING_OK: BOOL := FALSE;
	ALL_OFF: BOOL := FALSE;
	NOT_ALL_OFF: BOOL := FALSE;
	START_DELAY_ON: BOOL := FALSE;
	START_DELAY_OFF: BOOL := FALSE;
	STOP_DELAY_ON: BOOL := FALSE;
	STOP_DELAY_OFF: BOOL := FALSE;
	ENABLE_TIMER_ON: BOOL := FALSE;
	ENABLE_TIMER_OFF: BOOL := FALSE;
	BEEN_RUNNING_OK_LATCH: RS;
	ALL_OFF_LATCH: RS;
	START_DELAY_TON: TON;
	STOP_DELAY_TON: TON;
	STOPPED: INT;
END_VAR
VAR_INPUT
	ENABLE: BOOL := FALSE;
	STATUS: BOOL := FALSE;
	FIRE: BOOL := FALSE;
END_VAR
VAR_OUTPUT
	STATE: ET_9STATE_MONITORING := 9;
END_VAR

(* 
Version 1.0
Last Updated: 28/01/2020

9 States Monitoring. Value from 0 to 9
	STOPPED := 0,
	RUNNING := 1,
	STARTING := 2,
	STOPPING := 3,
	START_FAIL := 4,
	STOP_FAIL := 5,
	UNEXPECTED_START := 6,
	UNEXPECTED_STOP := 7,
	FIRE_STOP := 8,
	UNKNOWN := 9
*)

ENABLE_OFF := (ENABLE = FALSE);
ENABLE_ON := (ENABLE = TRUE);
STATUS_ON := (STATUS = TRUE);
STATUS_OFF := (STATUS = FALSE);
FIRE_ON := (FIRE = TRUE);
FIRE_OFF := (FIRE = FALSE);

BEEN_RUNNING_OK_LATCH(SET := ENABLE_ON AND STATUS_ON, RESET1 := ENABLE_OFF);
BEEN_RUNNING_OK := BEEN_RUNNING_OK_LATCH.Q1;

ALL_OFF_LATCH(SET := ENABLE_OFF AND STATUS_OFF, RESET1 := ENABLE_ON);
ALL_OFF := ALL_OFF_LATCH.Q1;

START_DELAY_TON(IN := ENABLE_ON, PT := T#30S);
START_DELAY_ON := START_DELAY_TON.Q;

STOP_DELAY_TON(IN := ENABLE_OFF, PT := T#30S);
STOP_DELAY_ON := STOP_DELAY_TON.Q;

ENABLE_TIMER_ON := ((START_DELAY_TON.ET < T#30S AND ENABLE_ON) OR (STOP_DELAY_TON.ET < T#30S AND ENABLE_OFF));

START_DELAY_OFF := NOT START_DELAY_ON;
STOP_DELAY_OFF := NOT STOP_DELAY_ON;
ENABLE_TIMER_OFF := NOT ENABLE_TIMER_ON;
NOT_BEEN_RUNNING_OK := NOT BEEN_RUNNING_OK;
NOT_ALL_OFF := NOT ALL_OFF;

IF (ENABLE_ON AND STATUS_OFF AND FIRE_ON) THEN
	STATE := ET_9STATE_MONITORING.FIRE_STOP;
ELSIF (ENABLE_OFF AND STATUS_ON AND STOP_DELAY_ON AND NOT_BEEN_RUNNING_OK AND NOT_ALL_OFF) THEN
	STATE := ET_9STATE_MONITORING.STOP_FAIL;
ELSIF (ENABLE_ON AND STATUS_OFF AND START_DELAY_ON AND NOT_BEEN_RUNNING_OK AND NOT_ALL_OFF) THEN
	STATE := ET_9STATE_MONITORING.START_FAIL;
ELSIF (ENABLE_OFF AND STATUS_ON AND ENABLE_TIMER_OFF AND STOP_DELAY_ON AND ENABLE_TIMER_OFF AND ALL_OFF) THEN
	STATE := ET_9STATE_MONITORING.UNEXPECTED_START;
ELSIF (ENABLE_ON AND STATUS_OFF AND START_DELAY_ON AND FIRE_OFF AND ENABLE_TIMER_OFF AND BEEN_RUNNING_OK AND NOT_ALL_OFF) THEN
	STATE := ET_9STATE_MONITORING.UNEXPECTED_STOP;
ELSIF (ENABLE_OFF AND STATUS_ON AND ENABLE_TIMER_ON AND STOP_DELAY_OFF AND FIRE_OFF) THEN
	STATE := ET_9STATE_MONITORING.STOPPING;
ELSIF (ENABLE_ON AND STATUS_ON) THEN
	STATE := ET_9STATE_MONITORING.RUNNING;
ELSIF (ENABLE_ON AND STATUS_OFF AND ENABLE_TIMER_ON AND START_DELAY_OFF AND FIRE_OFF) THEN
	STATE := ET_9STATE_MONITORING.STARTING;
ELSIF (ENABLE_OFF AND STATUS_OFF) THEN
	STATE := ET_9STATE_MONITORING.STOPPED;
ELSE
	STATE := ET_9STATE_MONITORING.UNKNOWN;
END_IF;

END_FUNCTION_BLOCK

// DCCM_PLC_3/Application/FBs/FB_DEPROX_SP
FUNCTION_BLOCK FB_DEPROX_SP
VAR_INPUT
	RM1: INT;
	RM2: INT;
	RM3: INT;
	RM4: INT;
	ONE_RM_SP: REAL;
	TWO_RM_SP: REAL;
	FOUR_RM_SP: REAL;
END_VAR
VAR_OUTPUT
	VP_SP: REAL;
	RM_TOTAL: REAL;
END_VAR
VAR_INPUT
	NORMAL_SP: REAL;
END_VAR
VAR
	DRM1: BOOL;
	DRM2: BOOL;
	DRM3: BOOL;
	DRM4: BOOL;
END_VAR

IF(RM1 = 0)THEN
	DRM1 := TRUE;
ELSE
	DRM1 := FALSE;

END_IF;
IF(RM2 = 0) THEN
	DRM2 := TRUE;
ELSE 
	DRM2 := FALSE;
END_IF;

IF(RM3 = 0) THEN
	DRM3 := TRUE;
ELSE
	DRM3 := FALSE;
END_IF;
IF(RM4 = 0) THEN
	DRM4 := TRUE;
ELSE
	DRM4 := FALSE;
END_IF;

RM_TOTAL := TO_REAL(DRM1) + TO_REAL(DRM2) + TO_REAL(DRM3) + TO_REAL(DRM4) ;
//IF (RM1 = TRUE AND RM2 = FALSE AND RM3 = FALSE AND RM4 = FALSE)
IF(RM_TOTAL = 0) THEN
	VP_SP := NORMAL_SP;
ELSIF(RM_TOTAL = 1) THEN
	VP_SP := ONE_RM_SP;
ELSIF(RM_TOTAL = 2 OR RM_TOTAL = 3) THEN
	VP_SP := TWO_RM_SP;
ELSIF(RM_TOTAL = 4) THEN
	VP_SP := FOUR_RM_SP;
	
END_IF;

END_FUNCTION_BLOCK

// DCCM_PLC_3/Application/FBs/MAN_AUTO_STS
FUNCTION_BLOCK MAN_AUTO_STS
VAR_INPUT
	MAN_SW: BOOL;
	AUTO_SW: BOOL;
END_VAR
VAR_OUTPUT
	STS: INT;
END_VAR

IF (MAN_SW = TRUE AND AUTO_SW = FALSE) THEN
	STS := 2;
ELSIF (AUTO_SW = TRUE AND MAN_SW = FALSE) THEN
	STS := 1;
ELSIF (AUTO_SW = FALSE AND MAN_SW = FALSE) THEN
	STS := 0;
ELSE
	STS := 3;
	
END_IF;

END_FUNCTION_BLOCK

// DCCM_PLC_3/Application/AHU_DAMPER_CONTROL
PROGRAM AHU_DAMPER_CONTROL
VAR
	AHU_RAD_SP: INT;
	LINEAR_0: LINEAR;
	LINEAR_1: LINEAR;
	A: BOOL;
	LINEAR_2: LINEAR;
	B: BOOL;
	TON_0: TON;
	TON_1: TON;
	TON_2: TON;
	TON_3: TON;
	TON_4: TON;
	TON_5: TON;
END_VAR

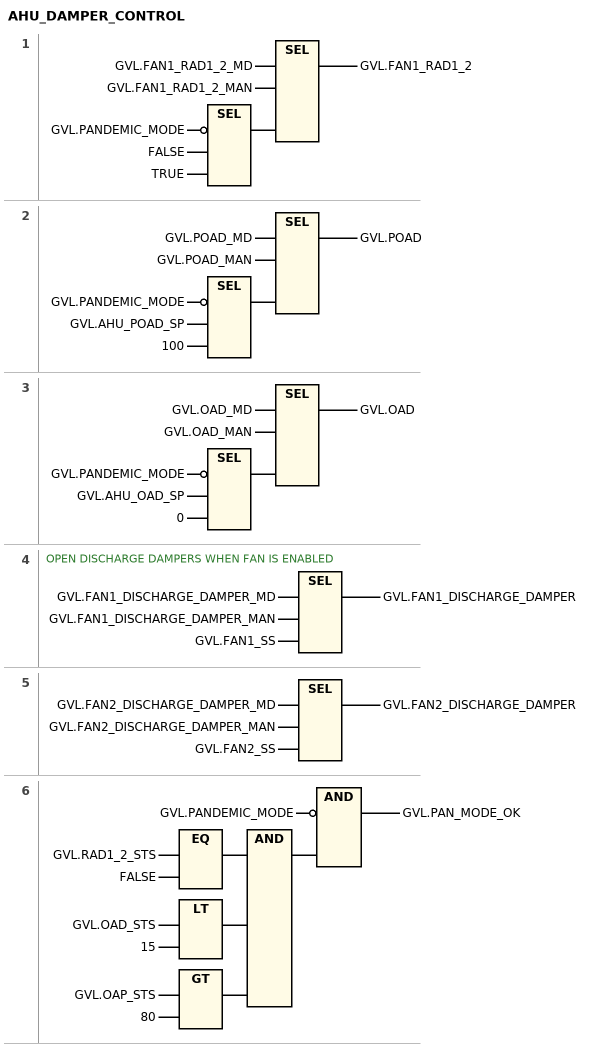
// NETWORK 1
GVL.FAN1_RAD1_2 := SEL(GVL.FAN1_RAD1_2_MD, GVL.FAN1_RAD1_2_MAN, SEL(NOT GVL.PANDEMIC_MODE, FALSE, TRUE));

// NETWORK 2
GVL.POAD := SEL(GVL.POAD_MD, GVL.POAD_MAN, SEL(NOT GVL.PANDEMIC_MODE, GVL.AHU_POAD_SP, 100));

// NETWORK 3
GVL.OAD := SEL(GVL.OAD_MD, GVL.OAD_MAN, SEL(NOT GVL.PANDEMIC_MODE, GVL.AHU_OAD_SP, 0));

// NETWORK 4
// OPEN DISCHARGE DAMPERS WHEN FAN IS ENABLED
GVL.FAN1_DISCHARGE_DAMPER := SEL(GVL.FAN1_DISCHARGE_DAMPER_MD, GVL.FAN1_DISCHARGE_DAMPER_MAN, GVL.FAN1_SS);

// NETWORK 5
GVL.FAN2_DISCHARGE_DAMPER := SEL(GVL.FAN2_DISCHARGE_DAMPER_MD, GVL.FAN2_DISCHARGE_DAMPER_MAN, GVL.FAN2_SS);

// NETWORK 6
GVL.PAN_MODE_OK := NOT GVL.PANDEMIC_MODE AND (GVL.RAD1_2_STS = FALSE AND GVL.OAD_STS < 15 AND GVL.OAP_STS > 80);

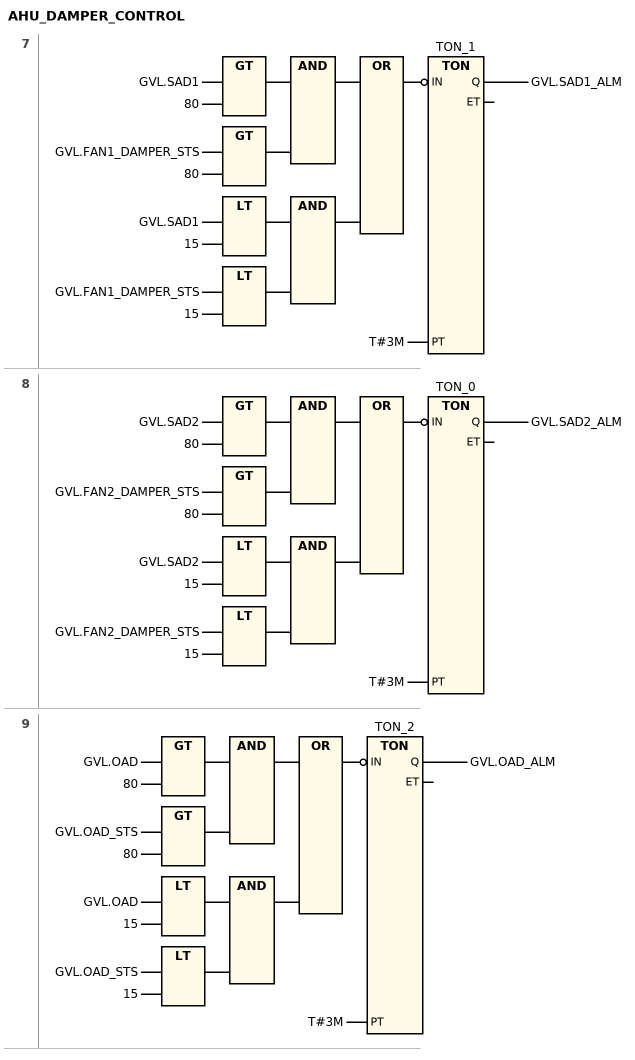
// NETWORK 7
TON_1(IN := NOT (GVL.SAD1 > 80 AND GVL.FAN1_DAMPER_STS > 80 OR GVL.SAD1 < 15 AND GVL.FAN1_DAMPER_STS < 15), PT := T#3M); // TON
GVL.SAD1_ALM := TON_1.Q;

// NETWORK 8
TON_0(IN := NOT (GVL.SAD2 > 80 AND GVL.FAN2_DAMPER_STS > 80 OR GVL.SAD2 < 15 AND GVL.FAN2_DAMPER_STS < 15), PT := T#3M); // TON
GVL.SAD2_ALM := TON_0.Q;

// NETWORK 9
TON_2(IN := NOT (GVL.OAD > 80 AND GVL.OAD_STS > 80 OR GVL.OAD < 15 AND GVL.OAD_STS < 15), PT := T#3M); // TON
GVL.OAD_ALM := TON_2.Q;

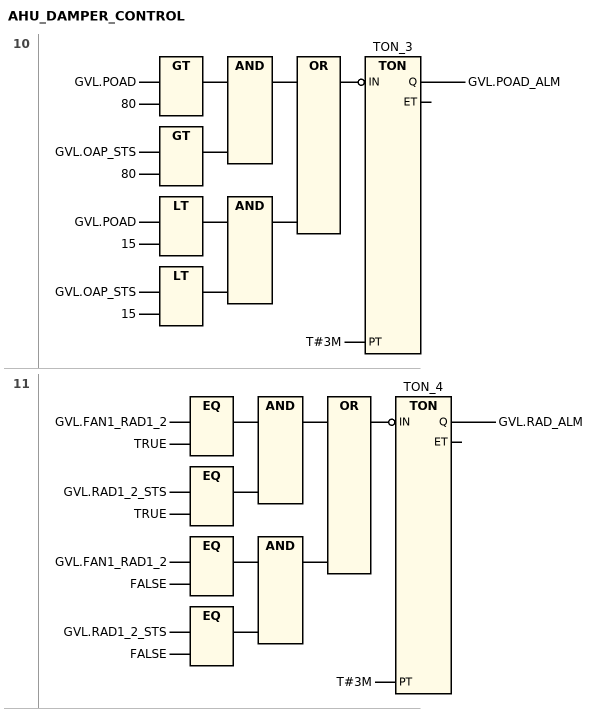
// NETWORK 10
TON_3(IN := NOT (GVL.POAD > 80 AND GVL.OAP_STS > 80 OR GVL.POAD < 15 AND GVL.OAP_STS < 15), PT := T#3M); // TON
GVL.POAD_ALM := TON_3.Q;

// NETWORK 11
TON_4(IN := NOT (GVL.FAN1_RAD1_2 = TRUE AND GVL.RAD1_2_STS = TRUE OR GVL.FAN1_RAD1_2 = FALSE AND GVL.RAD1_2_STS = FALSE), PT := T#3M); // TON
GVL.RAD_ALM := TON_4.Q;

END_PROGRAM

// DCCM_PLC_3/Application/AHU_TEMP_CONTROL
PROGRAM AHU_TEMP_CONTROL

VAR
	FB_MAX4_0: FB_MAX4;
	SATSP_CALC_0: SATSP_CALC;
	FB_HEATING_OR_COOLING_0: FB_HEATING_OR_COOLING;
	HEAT: BOOL;
	COOL: BOOL;
	HV_PID: PID;
	CV_PID: PID;
	HV_P: REAL := 2.5;
	HV_I: REAL := 12.5;
	CV_P: REAL := -2.5;
	CV_I: REAL := 12.5;
	LINEAR_0: LINEAR;
	A: BOOL;
	LINEAR_1: LINEAR;
	B: BOOL;
END_VAR

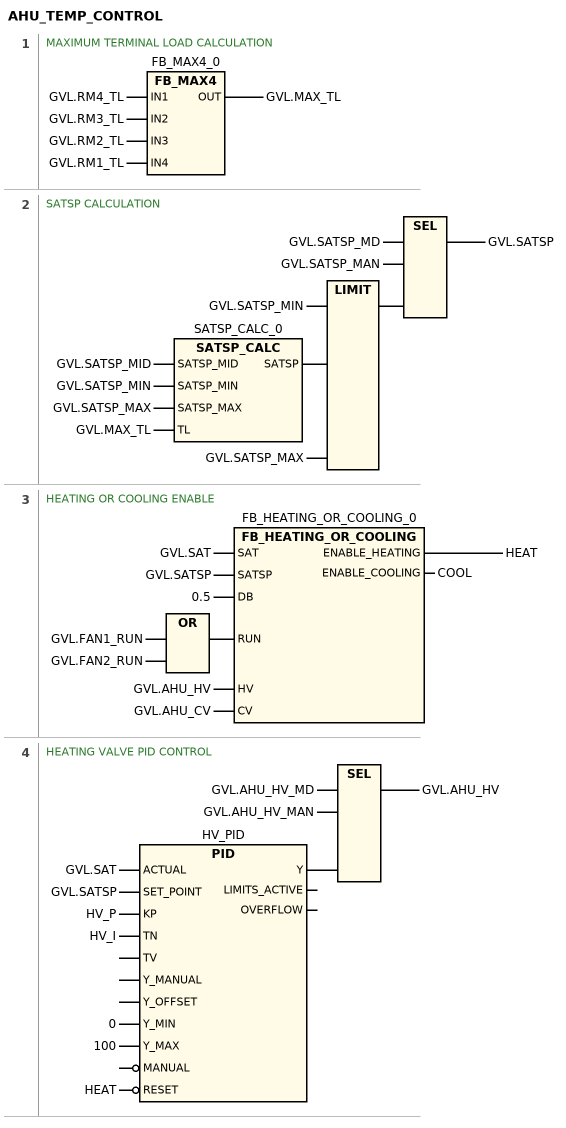
// NETWORK 1
// MAXIMUM TERMINAL LOAD CALCULATION
FB_MAX4_0(IN1 := GVL.RM4_TL, IN2 := GVL.RM3_TL, IN3 := GVL.RM2_TL, IN4 := GVL.RM1_TL); // FB_MAX4
GVL.MAX_TL := FB_MAX4_0.OUT;

// NETWORK 2
// SATSP CALCULATION
SATSP_CALC_0(
    SATSP_MID := GVL.SATSP_MID,
    SATSP_MIN := GVL.SATSP_MIN,
    SATSP_MAX := GVL.SATSP_MAX,
    TL := GVL.MAX_TL); // SATSP_CALC
GVL.SATSP := SEL(GVL.SATSP_MD, GVL.SATSP_MAN, LIMIT(GVL.SATSP_MIN, SATSP_CALC_0.SATSP, GVL.SATSP_MAX));

// NETWORK 3
// HEATING OR COOLING ENABLE
FB_HEATING_OR_COOLING_0(
    SAT := GVL.SAT,
    SATSP := GVL.SATSP,
    DB := 0.5,
    RUN := GVL.FAN1_RUN OR GVL.FAN2_RUN,
    HV := GVL.AHU_HV,
    CV := GVL.AHU_CV,
    ENABLE_COOLING => COOL); // FB_HEATING_OR_COOLING
HEAT := FB_HEATING_OR_COOLING_0.ENABLE_HEATING;

// NETWORK 4
// HEATING VALVE PID CONTROL
HV_PID(
    ACTUAL := GVL.SAT,
    SET_POINT := GVL.SATSP,
    KP := HV_P,
    TN := HV_I,
    Y_MIN := 0,
    Y_MAX := 100,
    RESET := NOT HEAT); // PID
GVL.AHU_HV := SEL(GVL.AHU_HV_MD, GVL.AHU_HV_MAN, HV_PID.Y);

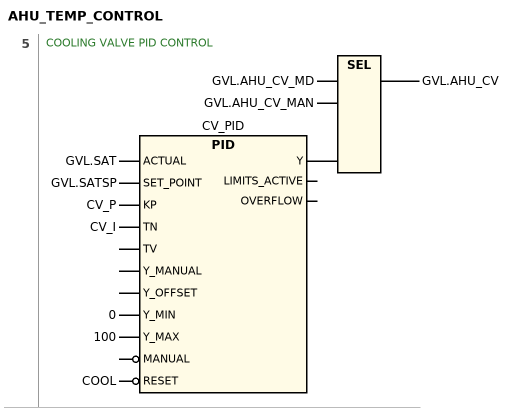
// NETWORK 5
// COOLING VALVE PID CONTROL
CV_PID(
    ACTUAL := GVL.SAT,
    SET_POINT := GVL.SATSP,
    KP := CV_P,
    TN := CV_I,
    Y_MIN := 0,
    Y_MAX := 100,
    RESET := NOT COOL); // PID
GVL.AHU_CV := SEL(GVL.AHU_CV_MD, GVL.AHU_CV_MAN, CV_PID.Y);

END_PROGRAM

// DCCM_PLC_3/Application/FBs/FB_MAX4
FUNCTION_BLOCK FB_MAX4
VAR_INPUT
	IN1: REAL;
	IN2: REAL;
	IN3: REAL;
	IN4: REAL;
END_VAR
VAR_OUTPUT
	OUT: REAL;
END_VAR

OUT := MAX(IN1, IN2, IN3, IN4);

END_FUNCTION_BLOCK

// DCCM_PLC_3/Application/FBs/SATSP_CALC
FUNCTION_BLOCK SATSP_CALC
VAR_INPUT
	SATSP_MID: REAL;
	SATSP_MIN: REAL;
	SATSP_MAX: REAL;
	TL: REAL;
END_VAR
VAR_OUTPUT
	SATSP: REAL;
END_VAR
VAR
	M: REAL;
END_VAR

IF TL > 0 THEN
	M := (SATSP_MID - SATSP_MIN) / 100.0;
	SATSP := SATSP_MId - (M * (TL));
ELSIF TL < 0 THEN
	M := (SATSP_MAX - SATSP_MID) / 100.0;
	SATSP := (M * ABS(TL)) + SATSP_MID;
ELSE
	SATSP := SATSP_MID;
END_IF;

END_FUNCTION_BLOCK

// DCCM_PLC_3/Application/FBs/FB_HEATING_OR_COOLING
FUNCTION_BLOCK FB_HEATING_OR_COOLING
VAR_INPUT
	SAT: REAL;
	SATSP: REAL;
	DB: REAL;
END_VAR
VAR_OUTPUT
	ENABLE_HEATING: BOOL;
	ENABLE_COOLING: BOOL;
END_VAR
VAR_INPUT
	RUN: BOOL;
	HV: REAL;
	CV: REAL;
END_VAR

IF (SAT >= (SATSP + DB) AND RUN AND HV = 0) THEN
	ENABLE_COOLING := TRUE; 
    ENABLE_HEATING := FALSE;
ELSIF (SAT <= (SATSP - DB) AND RUN AND CV = 0) THEN
	ENABLE_COOLING := FALSE;
    ENABLE_HEATING := TRUE;
ELSE
	ENABLE_COOLING := FALSE; 
    ENABLE_HEATING := FALSE;	
END_IF

END_FUNCTION_BLOCK

// DCCM_PLC_3/Application/RM1_TERMINAL_LOAD
PROGRAM RM1_TERMINAL_LOAD
VAR
	HEAT_TL_PID: PID;
	COOL_TL_PID: PID;
	HEAT_P: REAL := 2.5;
	HEAT_I: REAL := 12.5;
	HEAT_TL: REAL;
	COOL_P: REAL := -2.5;
	COOL_I: REAL := 12.5;
	COOL_TL: REAL;
	TERMINAL_LOAD_0: TERMINAL_LOAD;
END_VAR

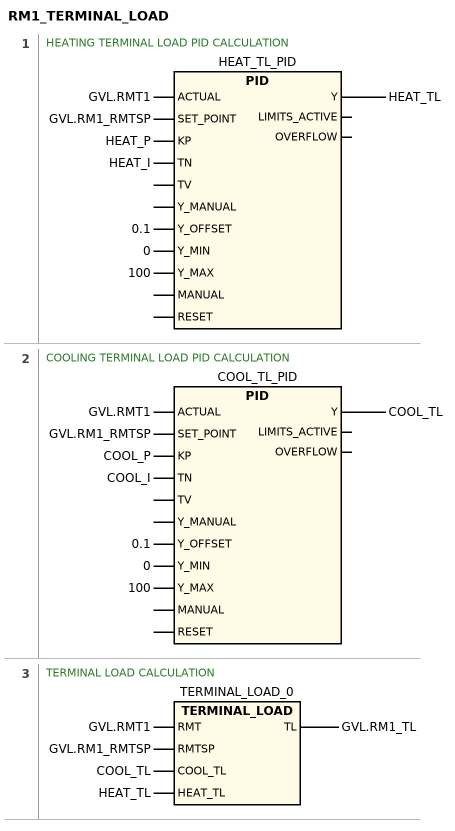
// NETWORK 1
// HEATING TERMINAL LOAD PID CALCULATION
HEAT_TL_PID(
    ACTUAL := GVL.RMT1,
    SET_POINT := GVL.RM1_RMTSP,
    KP := HEAT_P,
    TN := HEAT_I,
    Y_OFFSET := 0.1,
    Y_MIN := 0,
    Y_MAX := 100); // PID
HEAT_TL := HEAT_TL_PID.Y;

// NETWORK 2
// COOLING TERMINAL LOAD PID CALCULATION
COOL_TL_PID(
    ACTUAL := GVL.RMT1,
    SET_POINT := GVL.RM1_RMTSP,
    KP := COOL_P,
    TN := COOL_I,
    Y_OFFSET := 0.1,
    Y_MIN := 0,
    Y_MAX := 100); // PID
COOL_TL := COOL_TL_PID.Y;

// NETWORK 3
// TERMINAL LOAD CALCULATION
TERMINAL_LOAD_0(RMT := GVL.RMT1, RMTSP := GVL.RM1_RMTSP, COOL_TL := COOL_TL, HEAT_TL := HEAT_TL); // TERMINAL_LOAD
GVL.RM1_TL := TERMINAL_LOAD_0.TL;

END_PROGRAM

// DCCM_PLC_3/Application/FBs/TERMINAL_LOAD
FUNCTION_BLOCK TERMINAL_LOAD
VAR_INPUT
	RMT: REAL;
	RMTSP: REAL;
END_VAR
VAR_OUTPUT
	TL: REAL;
END_VAR
VAR_INPUT
	COOL_TL: REAL;
	HEAT_TL: REAL;
END_VAR

IF (RMTSP > RMT) THEN
	TL := (-1.0 * HEAT_TL);
ELSE
	TL := COOL_TL;	
END_IF;

END_FUNCTION_BLOCK

// DCCM_PLC_3/Application/RM2_TERMINAL_LOAD
PROGRAM RM2_TERMINAL_LOAD
VAR
	HEAT_TL_PID: PID;
	COOL_TL_PID: PID;
	HEAT_P: REAL := 2.5;
	HEAT_I: REAL := 12.5;
	HEAT_TL: REAL;
	COOL_P: REAL := -2.5;
	COOL_I: REAL := 12.5;
	COOL_TL: REAL;
	TERMINAL_LOAD_0: TERMINAL_LOAD;
END_VAR

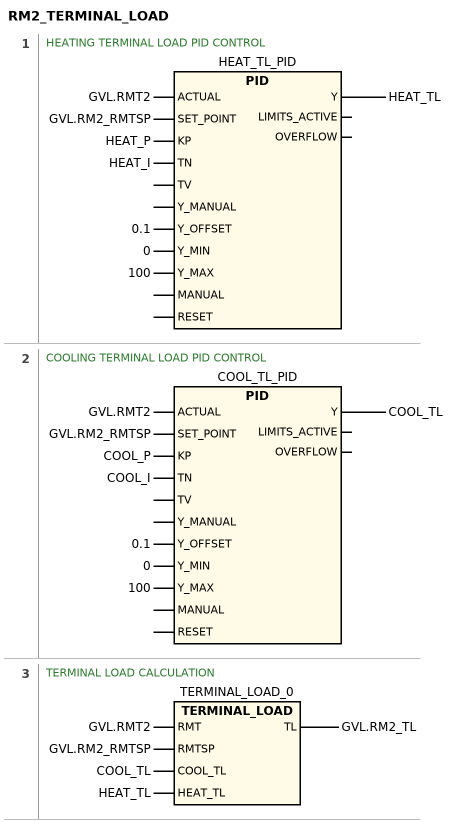
// NETWORK 1
// HEATING TERMINAL LOAD PID CONTROL
HEAT_TL_PID(
    ACTUAL := GVL.RMT2,
    SET_POINT := GVL.RM2_RMTSP,
    KP := HEAT_P,
    TN := HEAT_I,
    Y_OFFSET := 0.1,
    Y_MIN := 0,
    Y_MAX := 100); // PID
HEAT_TL := HEAT_TL_PID.Y;

// NETWORK 2
// COOLING TERMINAL LOAD PID CONTROL
COOL_TL_PID(
    ACTUAL := GVL.RMT2,
    SET_POINT := GVL.RM2_RMTSP,
    KP := COOL_P,
    TN := COOL_I,
    Y_OFFSET := 0.1,
    Y_MIN := 0,
    Y_MAX := 100); // PID
COOL_TL := COOL_TL_PID.Y;

// NETWORK 3
// TERMINAL LOAD CALCULATION
TERMINAL_LOAD_0(RMT := GVL.RMT2, RMTSP := GVL.RM2_RMTSP, COOL_TL := COOL_TL, HEAT_TL := HEAT_TL); // TERMINAL_LOAD
GVL.RM2_TL := TERMINAL_LOAD_0.TL;

END_PROGRAM

// DCCM_PLC_3/Application/RM3_TERMINAL_LOAD
PROGRAM RM3_TERMINAL_LOAD
VAR
	HEAT_TL_PID: PID;
	COOL_TL_PID: PID;
	HEAT_P: REAL := 2.5;
	HEAT_I: REAL := 12.5;
	HEAT_TL: REAL;
	COOL_P: REAL := -2.5;
	COOL_I: REAL := 12.5;
	COOL_TL: REAL;
	TERMINAL_LOAD_0: TERMINAL_LOAD;
END_VAR

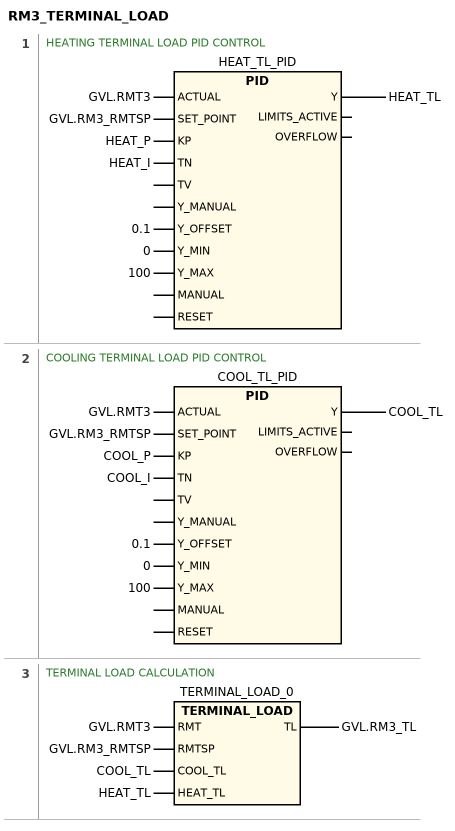
// NETWORK 1
// HEATING TERMINAL LOAD PID CONTROL
HEAT_TL_PID(
    ACTUAL := GVL.RMT3,
    SET_POINT := GVL.RM3_RMTSP,
    KP := HEAT_P,
    TN := HEAT_I,
    Y_OFFSET := 0.1,
    Y_MIN := 0,
    Y_MAX := 100); // PID
HEAT_TL := HEAT_TL_PID.Y;

// NETWORK 2
// COOLING TERMINAL LOAD PID CONTROL
COOL_TL_PID(
    ACTUAL := GVL.RMT3,
    SET_POINT := GVL.RM3_RMTSP,
    KP := COOL_P,
    TN := COOL_I,
    Y_OFFSET := 0.1,
    Y_MIN := 0,
    Y_MAX := 100); // PID
COOL_TL := COOL_TL_PID.Y;

// NETWORK 3
// TERMINAL LOAD CALCULATION
TERMINAL_LOAD_0(RMT := GVL.RMT3, RMTSP := GVL.RM3_RMTSP, COOL_TL := COOL_TL, HEAT_TL := HEAT_TL); // TERMINAL_LOAD
GVL.RM3_TL := TERMINAL_LOAD_0.TL;

END_PROGRAM

// DCCM_PLC_3/Application/RM4_TERMINAL_LOAD
PROGRAM RM4_TERMINAL_LOAD
VAR
	HEAT_TL_PID: PID;
	COOL_TL_PID: PID;
	HEAT_P: REAL := 2.5;
	HEAT_I: REAL := 12.5;
	HEAT_TL: REAL;
	COOL_P: REAL := -2.5;
	COOL_I: REAL := 12.5;
	COOL_TL: REAL;
	TERMINAL_LOAD_0: TERMINAL_LOAD;
END_VAR

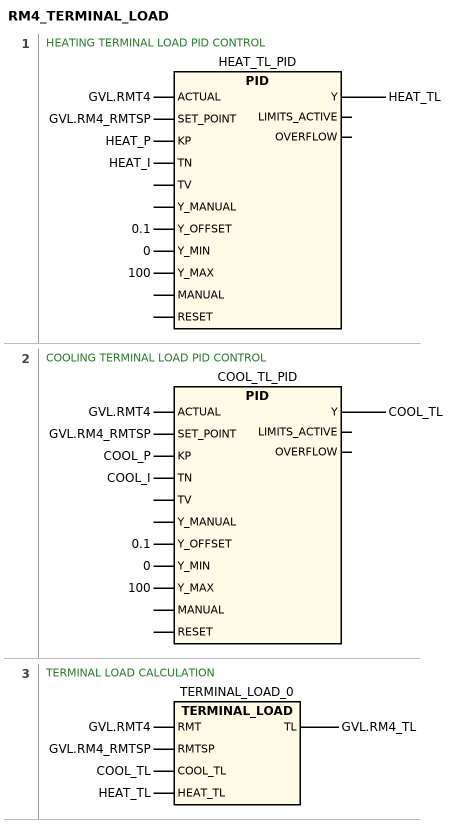
// NETWORK 1
// HEATING TERMINAL LOAD PID CONTROL
HEAT_TL_PID(
    ACTUAL := GVL.RMT4,
    SET_POINT := GVL.RM4_RMTSP,
    KP := HEAT_P,
    TN := HEAT_I,
    Y_OFFSET := 0.1,
    Y_MIN := 0,
    Y_MAX := 100); // PID
HEAT_TL := HEAT_TL_PID.Y;

// NETWORK 2
// COOLING TERMINAL LOAD PID CONTROL
COOL_TL_PID(
    ACTUAL := GVL.RMT4,
    SET_POINT := GVL.RM4_RMTSP,
    KP := COOL_P,
    TN := COOL_I,
    Y_OFFSET := 0.1,
    Y_MIN := 0,
    Y_MAX := 100); // PID
COOL_TL := COOL_TL_PID.Y;

// NETWORK 3
// TERMINAL LOAD CALCULATION
TERMINAL_LOAD_0(RMT := GVL.RMT4, RMTSP := GVL.RM4_RMTSP, COOL_TL := COOL_TL, HEAT_TL := HEAT_TL); // TERMINAL_LOAD
GVL.RM4_TL := TERMINAL_LOAD_0.TL;

END_PROGRAM

// DCCM_PLC_3/Application/TEST_VAR
PROGRAM TEST_VAR
VAR
	My_Read_Var: READ_VAR;
	Recieve_Buffer: ARRAY[0..3] OF INT;
	My_Addr_Table: ADDRESS;
	My_Addm: ADDM;
	My_Blink: BLINK;
	My_FLOAT: INT;
	lastValue: INT;
END_VAR

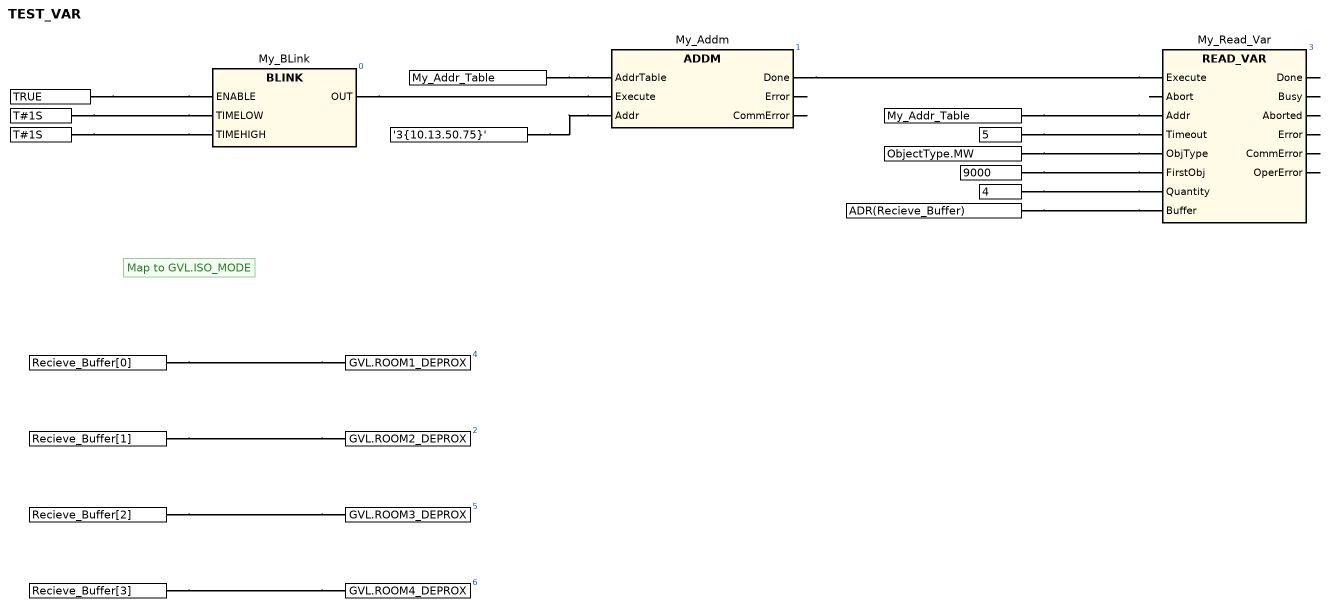
My_BLink(ENABLE := TRUE, TIMELOW := T#1S, TIMEHIGH := T#1S); // BLINK
My_Addm(AddrTable := My_Addr_Table, Execute := My_BLink.OUT, Addr := '3{10.13.50.75}'); // ADDM
GVL.ROOM2_DEPROX := Recieve_Buffer[1];
My_Read_Var(
    Execute := My_Addm.Done,
    Addr := My_Addr_Table,
    Timeout := 5,
    ObjType := ObjectType.MW,
    FirstObj := 9000,
    Quantity := 4,
    Buffer := ADR(Recieve_Buffer)); // READ_VAR
// Map to GVL.ISO_MODE
GVL.ROOM1_DEPROX := Recieve_Buffer[0];
GVL.ROOM3_DEPROX := Recieve_Buffer[2];
GVL.ROOM4_DEPROX := Recieve_Buffer[3];

END_PROGRAM

// DCCM_PLC_3/Application/SYSTEM_DATE_TIME
PROGRAM SYSTEM_DATE_TIME
VAR
	SysTimeRtcGetResult: UDINT;
	SYS_CLOCK: SysTimeRtc.RTS_SYSTIMEDATE;
END_VAR

//The following program initializes the system date time clock for the PLC. The date/time is subject to variance based on the temperature of the PLC, however this should not cause significant variance unless specific timing is required.
//For the sake of this project, the internal system clock is used for the duty change, tank turnover, etc. - Corey 21.07.2021

//Initializing the system date time
SysTimeRtc.SysTimeRtcConvertUtcToDate( dwTimestampUtc:= SysTimeRtc.SysTimeRtcGet( pResult:= SysTimeRtcGetResult ), pDate:= SYS_CLOCK );

//Updating the global variables for the date, hour and minute using the updated system time.
GVL.SYS_DAY := SYS_CLOCK.wDayOfWeek;
GVL.SYS_HOUR := SYS_CLOCK.wHour;
GVL.SYS_MINUTE := SYS_CLOCK.wMinute;

END_PROGRAM

// DCCM_PLC_3/Application/FBs/DUTY
FUNCTION_BLOCK DUTY
VAR_INPUT
	DUTY_MAN: BOOL;
	DUTY_MD: BOOL;
	TOGGLE: BOOL;
END_VAR
VAR_OUTPUT
	DUTY: BOOL;
END_VAR

IF (TOGGLE AND DUTY = TRUE AND DUTY_MD = FALSE) THEN
	DUTY := FALSE;
ELSIF (TOGGLE AND DUTY = FALSE AND DUTY_MD = FALSE) THEN
	DUTY := TRUE;
ELSE
	DUTY := DUTY_MAN;
END_IF

END_FUNCTION_BLOCK

// DCCM_PLC_3/Application/OUTPUT_MAPPING
PROGRAM OUTPUT_MAPPING
VAR
	BELIMO_OP: FB_0_10V_TO_2_10V_OUTPUT;
	LIN: LINEAR;
END_VAR

//MAPPING MEMORY WORDS TO HARDWARE OUTPUTS

qFAN1_SPD := TO_INT(GVL.FAN1_SPD) * 100;							//MODULE 1 TM3AM6 OUTPUT 0
qFAN2_SPD := TO_INT(GVL.FAN2_SPD) * 100;							//MODULE 1 TM3AM6 OUTPUT 1

//BELIMO_OP(IN_PRCT := TO_INT(GVL.AHU_CV));
//qAHU_HV := TO_INT(BELIMO_OP.OUT_PRCT * 100);								//MODULE 2 TM3AM6 OUTPUT 0
//BELIMO_OP(IN_PRCT := GVL.AHU_HV);
//qAHU_CV := TO_INT(BELIMO_OP.OUT_PRCT * 100);								//MODULE 2 TM3AM6 OUTPUT 1

//BELIMO_OP(IN_PRCT := GVL.OAD);
//qOAD1 := 10000 - TO_INT(BELIMO_OP.OUT_PRCT * 100);							//MODULE 3 TM3AM6 OUTPUT 0
//BELIMO_OP(IN_PRCT := GVL.POAD);
//qOAD2 := 10000 - TO_INT(BELIMO_OP.OUT_PRCT * 100);							//MODULE 3 TM3AM6 OUTPUT 1

LIN(INPUT := GVL.AHU_CV, X1 := 0, Y1 := 2000, X2 := 100, Y2 := 10000);
qAHU_CV := TO_INT(LIN.OUTPUT); 
LIN(INPUT := GVL.AHU_HV, X1 := 0, Y1 := 2000, X2 := 100, Y2 := 10000);
qAHU_HV := TO_INT(LIN.OUTPUT); 

LIN(INPUT := GVL.OAD, X1 := 0, Y1 := 10000, X2 := 100, Y2 := 2000);
qOAD1 := TO_INT(LIN.OUTPUT); 
LIN(INPUT := GVL.POAD, X1 := 0, Y1 := 10000, X2 := 100, Y2 := 2000);
qOAD2 := TO_INT(LIN.OUTPUT); 
//BELIMO_OP(IN_PRCT := GVL.SAD1);
//qSAD1 := 10000 - TO_INT(BELIMO_OP.OUT_PRCT * 100);							//MODULE 4 TM3AM6 OUTPUT 0
LIN(INPUT := GVL.SAD1, X1 := 0, Y1 := 10000, X2 := 100, Y2 := 2000);
qSAD1 := TO_INT(LIN.OUTPUT); 
LIN(INPUT := GVL.SAD2, X1 := 0, Y1 := 10000, X2 := 100, Y2 := 2000);
qSAD2 := TO_INT(LIN.OUTPUT); 							//MODULE 4 TM3AM6 OUTPUT 1

qFAN1_SS := GVL.FAN1_SS;											//MODULE 5 TM3DM24R OUTPUT 0
qFAN2_SS := GVL.FAN2_SS;											//MODULE 5 TM3DM24R OUTPUT 1
qFAN1_RAD1_2 := GVL.FAN1_RAD1_2;									//MODULE 5 TM3DM24R OUTPUT 2
qISO_NORMAL_MODE := GVL.ISO_NORMAL_MODE;							//MODULE 5 TM3DM24R OUTPUT 3

END_PROGRAM

// DCCM_PLC_3/Application/LIBRARY/FB_0_10V_TO_2_10V_OUTPUT
FUNCTION_BLOCK FB_0_10V_TO_2_10V_OUTPUT
VAR_OUTPUT
	/// 0-10V = 0-100%
	OUT_PRCT: REAL;
END_VAR
VAR_INPUT
	/// 2-10V = 0-100%
	IN_PRCT: REAL;
END_VAR

OUT_PRCT := ((IN_PRCT * 0.08) * 10);

END_FUNCTION_BLOCK

// DCCM_PLC_3/Application/SR_Main
PROGRAM SR_Main
VAR
END_VAR

// NETWORK 1

END_PROGRAM

// DCCM_PLC_3/Application/FBs/SB_HEATING_COOLING
FUNCTION_BLOCK SB_HEATING_COOLING
VAR_INPUT
	ENABLE_COOLING: BOOL;
	ENABLE_HEATING: BOOL;
	SATSP: REAL;
	COOLING_SP: REAL;
	HEATING_SP: REAL;
END_VAR
VAR_OUTPUT
	OUT: REAL;
END_VAR
VAR_INPUT
	OMODE: ET_OMODE;
END_VAR

IF (ENABLE_COOLING AND OMODE = ET_OMODE.SETBACK) THEN
	OUT := COOLING_SP;
ELSIF (ENABLE_HEATING AND OMODE = ET_OMODE.SETBACK) THEN
	OUT := HEATING_SP;
ELSE
	OUT := SATSP;
END_IF

END_FUNCTION_BLOCK

// DCCM_PLC_3/Application/FBs/FB_SETPOINT_MODE
FUNCTION_BLOCK FB_SETPOINT_MODE
VAR_INPUT
	OMODE: ET_OMODE;
	PMODE: ET_PMODE;
	DAY_SP: REAL;
	SETBACK_SP: REAL;
	PURGE_SP: REAL;
END_VAR
VAR_OUTPUT
	RESULT: REAL;
END_VAR

(*
//calculate set point based on plant mode and occupancy mode
	/*
	//occupancy mode
	UNOCC := 0,
	OP_START := 1,
	SCH := 2,
	AHRS := 3,
	MOT_DETECT := 4,
	REVERSE1 := 5,
	REVERSE2 := 6,
	SETBACK := 7,
	
	//plant mode
	OFF_NORMAL := 0,
	OFF_PCMS := 1,
	OFF_FIRE := 2,
	OFF_DMPRLCK := 3,
	OFF_DMPRRESET := 4,
	STARTUP := 5,
	RUN_PUR := 6,
	RUN_NORMAL := 7
	*/
*)

IF (PMODE = ET_PMODE.Purge) THEN
	RESULT := PURGE_SP;
ELSIF ((PMODE = ET_PMODE.RUN_NORMAL) OR (PMODE = ET_PMODE.Startup)) THEN
	IF (OMODE = ET_OMODE.SETBACK) THEN
		RESULT := SETBACK_SP;
	ELSIF(OMODE = ET_OMODE.UNOCC) THEN
		RESULT := 0.0;
	ELSE
		RESULT := DAY_SP;
	END_IF
ELSE
	RESULT := DAY_SP;
END_IF

END_FUNCTION_BLOCK

// DCCM_PLC_3/Application/FBs/FB_FLOATING_VALVE
FUNCTION_BLOCK FB_FLOATING_VALVE
VAR_INPUT
	VALVE_OUTPUT: REAL;
	VALVE_TIME: TIME;
END_VAR
VAR_OUTPUT
	VALVE_OPEN: BOOL;
	VALVE_CLOSE: BOOL;
END_VAR
VAR
	CURRENT_POS: REAL;
	MOVE_TIME: TIME;
	MOVE_POS: REAL;
	RS_0: RS;
	TON1: TON;
	OPEN_STOP: BOOL;
	TON2: TON;
	CLOSE_STOP: BOOL;
	RS_1: RS;
END_VAR

IF (VALVE_OUTPUT > CURRENT_POS) THEN
	MOVE_POS := VALVE_OUTPUT - CURRENT_POS;
 	MOVE_TIME := TO_TIME(TO_REAL(VALVE_TIME) * (MOVE_POS / 100)); 
	VALVE_OPEN := TRUE;
	TON1(IN := VALVE_OPEN, PT := MOVE_TIME);
	OPEN_STOP := TON1.Q;
	//RS_0(SET := VALVE_OPEN, RESET1 := OPEN_STOP);
	IF (OPEN_STOP = TRUE) THEN
		VALVE_OPEN := FALSE;
		CURRENT_POS := VALVE_OUTPUT;
	END_IF  
ELSIF (VALVE_OUTPUT < CURRENT_POS) THEN
	MOVE_POS := CURRENT_POS - VALVE_OUTPUT;
	MOVE_TIME := TO_TIME(TO_REAL(VALVE_TIME) * (MOVE_POS / 100));
	VALVE_CLOSE := TRUE;
	TON2(IN := VALVE_CLOSE, PT := MOVE_TIME);
	CLOSE_STOP := TON2.Q;
	//RS_1(SET := VALVE_OPEN, RESET1 := CLOSE_STOP);
	IF (CLOSE_STOP = TRUE) THEN
		VALVE_CLOSE := FALSE;
		CURRENT_POS := VALVE_OUTPUT;
	END_IF
ELSE
	VALVE_OPEN := FALSE;
	VALVE_CLOSE := FALSE;
END_IF

END_FUNCTION_BLOCK

// DCCM_PLC_3/Application/FBs/FB_OMODE
FUNCTION_BLOCK FB_OMODE
VAR_INPUT
	ENABLE_BY_TP: BOOL;
	ENABLE_BY_PIR: BOOL;
	ENABLE_BY_AHRS: BOOL;
	MODE: BOOL;
	OMODE_MANUAL: ET_OMODE;
	TPTYPE: BOOL;
END_VAR
VAR_OUTPUT
	OMODE: ET_OMODE;
END_VAR




IF (MODE) THEN
	IF (ENABLE_BY_TP) THEN				//AUTO MODE
		OMODE := ET_OMODE.SCH;
	ELSIF (ENABLE_BY_AHRS) THEN
		OMODE := ET_OMODE.AHRS;
	ELSIF (ENABLE_BY_PIR) THEN
		OMODE := ET_OMODE.MOTDETECT;
	ELSIF (TPTYPE) THEN
		OMODE := ET_OMODE.UNOCC;
	ELSE
		OMODE := ET_OMODE.SETBACK;
	END_IF
ELSE
	OMODE := OMODE_MANUAL;				//MANUAL MODE
END_IF

END_FUNCTION_BLOCK

// DCCM_PLC_3/Application/FBs/FB_PMODE
FUNCTION_BLOCK FB_PMODE
VAR_INPUT
	OMODE: ET_OMODE;
	IS_NOT_SMOKE: BOOL := TRUE;
	FIRE: BOOL;
	PCMS_SIGNAL: INT;
	PCMS_PRIMARY: INT;
	PCMS_MODE: BOOL := TRUE;
	IS_DAMPER_LOCK: BOOL;
	IS_DAMPER_RESET: BOOL;
	IS_PURGE_RUN: BOOL;
	IS_DAMPER_STARTED: BOOL;
	PMODE_MODE: BOOL := TRUE;
	PMODE_MANUAL: ET_PMODE;
END_VAR
VAR_OUTPUT
	AHU_ENABLE: BOOL;
	PMODE: ET_PMODE;
END_VAR

(*  
	Version 1.0
	Last modified: 15/8/2022
	Operating theater mode
	PLEASE USE  FOR OPERATING THEATER ONLY
	IT DOES NOT IMPLEMENT UNOCC, OP_START MODE
	
	OFF_NORMAL := 0,
	OFF_PCMS := 1,
	OFF_FIRE := 2,
	OFF_DMPRLCK := 3,
	OFF_RESET := 4,
	STARTUP := 5,
	RUN_PUR := 6,
	RUN_NORMAL := 7
*)


IF (PMODE_MODE) THEN
	IF (FIRE) THEN
		PMODE := ET_PMODE.OFF_Fire;
	ELSIF (IS_DAMPER_LOCK) THEN
		PMODE := ET_PMODE.OFF_DMPRLOCK;
	ELSIF ((ABS(PCMS_SIGNAL) >= ABS(PCMS_PRIMARY)) AND PCMS_MODE) THEN
		PMODE := ET_PMODE.OFF_PCMS;
	ELSIF (IS_DAMPER_RESET) THEN
		PMODE := ET_PMODE.OFF_RESET;
	ELSIF (IS_PURGE_RUN) THEN
		PMODE := ET_PMODE.Purge;
	ELSIF (IS_DAMPER_STARTED) THEN
		PMODE := ET_PMODE.RUN_NORMAL;
	END_IF
ELSE
	PMODE := PMODE_MANUAL;
END_IF;

AHU_ENABLE := (PMODE = ET_PMODE.Startup OR PMODE = ET_PMODE.Purge OR PMODE = ET_PMODE.RUN_NORMAL) AND IS_NOT_SMOKE = FALSE AND OMODE <> ET_OMODE.UNOCC;

END_FUNCTION_BLOCK

// DCCM_PLC_3/Application/FBs/FB_WATCHDOG
FUNCTION_BLOCK FB_WATCHDOG
VAR_OUTPUT
	LAST_VALUE: INT;
END_VAR
VAR_INPUT
	VALUE: INT;
END_VAR
VAR_OUTPUT
	TIMEOUT: BOOL;
END_VAR
VAR
	START_DELAY_TON: TON;
END_VAR

START_DELAY_TON(IN := (LAST_VALUE = VALUE), PT := T#120S);
TIMEOUT := START_DELAY_TON.Q;

LAST_VALUE := VALUE;

END_FUNCTION_BLOCK

// DCCM_PLC_3/Application/FBs/FB_DUTY_DUTY_STANDBY_PUMP_SPD
FUNCTION_BLOCK FB_DUTY_DUTY_STANDBY_PUMP_SPD
VAR_INPUT
	SPD_DEM: REAL;
	P1_FLT: BOOL;
	P2_FLT: BOOL;
	P3_FLT: BOOL;
	DUTY: INT;
END_VAR
VAR_OUTPUT
	PUMP1_SPD: REAL;
	PUMP2_SPD: REAL;
	PUMP3_SPD: REAL;
END_VAR

IF (P1_FLT = TRUE AND P2_FLT = TRUE AND P3_FLT = TRUE) THEN				// IF ALL PUMPS IN FAULT, REDUCE SPEED TO 0 FOR ALL PUMPS
	PUMP1_SPD := 0;
	PUMP2_SPD := 0;
	PUMP3_SPD := 0;
ELSIF (DUTY = 0 AND P1_FLT = FALSE AND P2_FLT = FALSE) THEN				//IF PUMP 1 DUTY
	PUMP1_SPD := LIMIT(0, SPD_DEM, 100);
	PUMP2_SPD := LIMIT(0, SPD_DEM - 100, 100);
	PUMP3_SPD := 0;
ELSIF (DUTY = 1 AND P2_FLT = FALSE AND P3_FLT = FALSE)THEN				//IF PUMP 2 DUTY
	PUMP2_SPD := LIMIT(0, SPD_DEM, 100);
	PUMP3_SPD := LIMIT(0, SPD_DEM - 100, 100);
	PUMP1_SPD := 0;
ELSIF(DUTY = 2 AND P3_FLT = FALSE AND P1_FLT = FALSE) THEN				//IF PUMP 3 DUTY
	PUMP3_SPD := LIMIT(0, SPD_DEM, 100);
	PUMP1_SPD := LIMIT(0, SPD_DEM - 100, 100);
	PUMP2_SPD := 0;	
ELSIF (DUTY = 0 AND P1_FLT = TRUE AND P2_FLT = FALSE) THEN				//IF PUMP 1 DUTY AND PUMP 1 IS IN FAULT
	PUMP3_SPD := LIMIT(0, SPD_DEM, 100);
	PUMP2_SPD := LIMIT(0, SPD_DEM - 100, 100);
	PUMP1_SPD := 0;
ELSIF (DUTY = 0 AND P1_FLT = FALSE AND P2_FLT = TRUE) THEN				// IF PUMP 1 DUTY AND PUMP 2 IS IN FAULT
	PUMP1_SPD := LIMIT(0, SPD_DEM, 100);
	PUMP3_SPD := LIMIT(0, SPD_DEM - 100, 100);
	PUMP2_SPD := 0;
ELSIF (DUTY = 0 AND P1_FLT = TRUE AND P2_FLT = TRUE) THEN				//IF PUMP 1 DUTY AND PUMP 1 & 2 ARE IN FAULT
	PUMP3_SPD := LIMIT(0, SPD_DEM, 100);
	PUMP1_SPD := 0;
	PUMP2_SPD := 0;
ELSIF (DUTY = 1 AND P2_FLT = TRUE AND P3_FLT = FALSE) THEN				//IF PUMP 2 DUTY AND PUMP 2 IS IN FAULT
	PUMP1_SPD := LIMIT(0, SPD_DEM, 100);
	PUMP3_SPD := LIMIT(0, SPD_DEM - 100, 100);
	PUMP2_SPD := 0;
ELSIF (DUTY = 1 AND P2_FLT = FALSE AND P3_FLT := TRUE) THEN				//IF PUMP 2 DUTY AND PUMP 3 IS IN FAULT
	PUMP2_SPD := LIMIT(0, SPD_DEM, 100);
	PUMP1_SPD := LIMIT(0, SPD_DEM - 100, 100);
	PUMP3_SPD := 0;
ELSIF (DUTY = 1 AND P2_FLT = TRUE AND P3_FLT := TRUE) THEN				//IF PUMP 2 DUTY AND PUMP 2 & 3 ARE IN FAULT
	PUMP1_SPD := LIMIT(0, SPD_DEM, 100);
	PUMP2_SPD := 0;
	PUMP3_SPD := 0;
ELSIF (DUTY = 2 AND P3_FLT = TRUE AND P1_FLT = FALSE) THEN				//IF PUMP 3 DUTY AND PUMP 3 IS IN FAULT 
	PUMP2_SPD := LIMIT(0, SPD_DEM, 100);
	PUMP1_SPD := LIMIT(0, SPD_DEM - 100, 100);
	PUMP3_SPD := 0;
ELSIF (DUTY = 2 AND P3_FLT = FALSE AND P1_FLT = TRUE) THEN				//IF PUMP 3 DUTY AND PUMP 1 IS IN FAULT
	PUMP3_SPD := LIMIT(0, SPD_DEM, 100);
	PUMP2_SPD := LIMIT(0, SPD_DEM - 100, 100);
	PUMP1_SPD := 0;
ELSIF (DUTY = 2 AND P3_FLT = TRUE AND P1_FLT = TRUE) THEN				//IF PUMP 3 DUTY AND PUMP 3 & 1 ARE IN FAULT
	PUMP2_SPD := LIMIT(0, SPD_DEM, 100);
	PUMP3_SPD := 0;
	PUMP1_SPD := 0;
END_IF

END_FUNCTION_BLOCK

// DCCM_PLC_3/Application/Library/FB_SETPOINT_RAMPING
FUNCTION_BLOCK FB_SETPOINT_RAMPING
VAR_INPUT
	INPUT: REAL;
	RAMPING_DOWN_TIME_SP: REAL := 10;
	RAMPING_UP_TIME_SP: REAL := 10;
END_VAR
VAR_OUTPUT
	OUTPUT: REAL := 0;
END_VAR
VAR
	TIMER: TON;
	INCREMENT: REAL;
	INPUT_MEMORY: REAL;
END_VAR

(* Set point Ramping up and down *)
IF (OUTPUT = 0) THEN
	OUTPUT := INPUT;
END_IF;

//find the incerement value
IF(INPUT <> INPUT_MEMORY) THEN 
	INPUT_MEMORY := INPUT;	
	IF (INPUT_MEMORY > OUTPUT) THEN
		INCREMENT := (INPUT_MEMORY - OUTPUT)/RAMPING_UP_TIME_SP;
	ELSIF (INPUT_MEMORY < OUTPUT) THEN
		INCREMENT := (INPUT_MEMORY - OUTPUT)/RAMPING_DOWN_TIME_SP;
	ELSE
		INCREMENT := 0;
	END_IF;
END_IF;


IF(INCREMENT <> 0) THEN
	TIMER(IN := NOT TIMER.Q, PT := T#1S);

	IF (TIMER.Q) THEN
		OUTPUT := OUTPUT + INCREMENT;
	END_IF;
	
	IF(OUTPUT > INPUT_MEMORY) AND (INCREMENT > 0) THEN
		//make sure that the output is not over than ouput
		INCREMENT := 0;
		OUTPUT := INPUT_MEMORY;
	ELSIF (OUTPUT < INPUT_MEMORY) AND (INCREMENT < 0) THEN
		//make sure that the output is not less than input
		INCREMENT := 0;
		OUTPUT := INPUT_MEMORY;
	END_IF;
END_IF;

END_FUNCTION_BLOCK

// DCCM_PLC_3/Application/LIBRARY/FB_PULSE_GENERATOR
FUNCTION_BLOCK FB_PULSE_GENERATOR
VAR_INPUT
	ENABLE: BOOL;
END_VAR
VAR_OUTPUT
	OUTPUT: BOOL;
END_VAR
VAR
	PULSESTATE: BOOL;
	PULSETIME: INT;
END_VAR


IF (ENABLE) THEN
	IF(PULSETIME > 100) THEN
		PULSESTATE := NOT PULSESTATE;
		PULSETIME := 0;
	END_IF;
	IF (PULSETIME < 0) THEN
		PULSETIME := 0;
	END_IF;
ELSE
	PULSESTATE := FALSE;
	PULSETIME := 0;
END_IF;

PULSETIME := PULSETIME +1;

OUTPUT := PULSESTATE;

END_FUNCTION_BLOCK
